LIN {X 0.129,Y -485.404,Z 1314.545,A 0.000,B 0.000,C 90.000,E1 98.106} C_DIS
LIN {X -0.160,Y -484.743,Z 1314.542,A 0.000,B 0.000,C 90.000,E1 97.644} C_DIS
LIN {X 0.035,Y -482.997,Z 1314.540,A 0.000,B 0.000,C 90.000,E1 97.125} C_DIS
LIN {X -0.080,Y -481.617,Z 1314.538,A 0.000,B 0.000,C 90.000,E1 96.891} C_DIS
LIN {X 0.196,Y -468.676,Z 1314.528,A 0.000,B 0.000,C 90.000,E1 95.106} C_DIS
LIN {X -0.021,Y -455.031,Z 1314.517,A 0.000,B 0.000,C 90.000,E1 93.094} C_DIS
LIN {X -0.140,Y -441.662,Z 1314.506,A 0.000,B 0.000,C 90.000,E1 91.031} C_DIS
LIN {X 0.133,Y -422.329,Z 1314.486,A 0.000,B 0.000,C 90.000,E1 87.535} C_DIS
LIN {X 0.147,Y -410.730,Z 1314.474,A 0.000,B 0.000,C 90.000,E1 85.355} C_DIS
LIN {X -0.079,Y -400.504,Z 1314.464,A 0.000,B 0.000,C 90.000,E1 83.451} C_DIS
LIN {X -0.116,Y -390.001,Z 1314.453,A 0.000,B 0.000,C 90.000,E1 81.489} C_DIS
LIN {X 0.060,Y -382.304,Z 1314.445,A 0.000,B 0.000,C 90.000,E1 80.038} C_DIS
LIN {X 0.190,Y -372.725,Z 1314.435,A 0.000,B 0.000,C 90.000,E1 78.285} C_DIS
LIN {X 0.196,Y -361.322,Z 1314.424,A 0.000,B 0.000,C 90.000,E1 76.228} C_DIS
LIN {X 0.053,Y -349.781,Z 1314.412,A 0.000,B 0.000,C 90.000,E1 74.157} C_DIS
LIN {X -0.138,Y -339.831,Z 1314.402,A 0.000,B 0.000,C 90.000,E1 72.362} C_DIS
LIN {X -0.137,Y -326.623,Z 1314.388,A 0.000,B 0.000,C 90.000,E1 69.880} C_DIS
LIN {X 0.035,Y -310.894,Z 1314.370,A 0.000,B 0.000,C 90.000,E1 66.666} C_DIS
LIN {X 0.081,Y -297.924,Z 1314.354,A 0.000,B 0.000,C 90.000,E1 63.717} C_DIS
LIN {X 0.082,Y -290.234,Z 1314.343,A 0.000,B 0.000,C 90.000,E1 61.719} C_DIS
LIN {X -0.050,Y -282.326,Z 1314.330,A 0.000,B 0.000,C 90.000,E1 59.380} C_DIS
LIN {X 0.051,Y -272.343,Z 1314.311,A 0.000,B 0.000,C 90.000,E1 55.928} C_DIS
LIN {X 0.059,Y -263.219,Z 1314.291,A 0.000,B 0.000,C 90.000,E1 52.431} C_DIS
LIN {X -0.081,Y -256.340,Z 1314.276,A 0.000,B 0.000,C 90.000,E1 49.622} C_DIS
LIN {X -0.074,Y -249.674,Z 1314.260,A 0.000,B 0.000,C 90.000,E1 46.743} C_DIS
LIN {X -0.083,Y -241.652,Z 1314.239,A 0.000,B 0.000,C 90.000,E1 43.095} C_DIS
LIN {X 0.031,Y -234.237,Z 1314.219,A 0.000,B 0.000,C 90.000,E1 39.358} C_DIS
LIN {X 0.013,Y -227.695,Z 1314.198,A 0.000,B 0.000,C 90.000,E1 35.598} C_DIS
LIN {X -0.050,Y -222.189,Z 1314.177,A 0.000,B 0.000,C 90.000,E1 31.799} C_DIS
LIN {X 0.121,Y -217.581,Z 1314.155,A 0.000,B 0.000,C 90.000,E1 27.897} C_DIS
LIN {X 0.034,Y -213.697,Z 1314.134,A 0.000,B 0.000,C 90.000,E1 24.027} C_DIS
LIN {X -0.036,Y -210.214,Z 1314.112,A 0.000,B 0.000,C 90.000,E1 20.120} C_DIS
LIN {X 0.080,Y -207.058,Z 1314.090,A 0.000,B 0.000,C 90.000,E1 16.134} C_DIS
LIN {X 0.003,Y -204.286,Z 1314.068,A 0.000,B 0.000,C 90.000,E1 12.175} C_DIS
LIN {X 0.056,Y -201.522,Z 1314.041,A 0.000,B 0.000,C 90.000,E1 7.352} C_DIS
LIN {X 0.006,Y -199.312,Z 1314.005,A 0.000,B 0.000,C 90.000,E1 0.917} C_DIS
LIN {X 0.017,Y -199.411,Z 1313.957,A 0.000,B 0.000,C 90.000,E1 352.243} C_DIS
LIN {X 0.019,Y -201.511,Z 1313.926,A 0.000,B 0.000,C 90.000,E1 346.589} C_DIS
LIN {X 0.030,Y -204.619,Z 1313.899,A 0.000,B 0.000,C 90.000,E1 341.764} C_DIS
LIN {X 0.046,Y -209.021,Z 1313.872,A 0.000,B 0.000,C 90.000,E1 336.975} C_DIS
LIN {X -0.054,Y -213.620,Z 1313.850,A 0.000,B 0.000,C 90.000,E1 333.050} C_DIS
LIN {X 0.001,Y -219.164,Z 1313.828,A 0.000,B 0.000,C 90.000,E1 329.125} C_DIS
LIN {X 0.001,Y -225.693,Z 1313.807,A 0.000,B 0.000,C 90.000,E1 325.261} C_DIS
LIN {X -0.020,Y -233.132,Z 1313.786,A 0.000,B 0.000,C 90.000,E1 321.457} C_DIS
LIN {X -0.056,Y -241.637,Z 1313.765,A 0.000,B 0.000,C 90.000,E1 317.715} C_DIS
LIN {X 0.140,Y -250.446,Z 1313.747,A 0.000,B 0.000,C 90.000,E1 314.352} C_DIS
LIN {X 0.079,Y -259.281,Z 1313.730,A 0.000,B 0.000,C 90.000,E1 311.472} C_DIS
LIN {X 0.033,Y -268.239,Z 1313.717,A 0.000,B 0.000,C 90.000,E1 308.991} C_DIS
LIN {X 0.134,Y -276.833,Z 1313.705,A 0.000,B 0.000,C 90.000,E1 306.870} C_DIS
LIN {X 0.035,Y -288.162,Z 1313.692,A 0.000,B 0.000,C 90.000,E1 304.485} C_DIS
LIN {X 0.018,Y -300.990,Z 1313.679,A 0.000,B 0.000,C 90.000,E1 302.133} C_DIS
LIN {X 0.100,Y -309.231,Z 1313.671,A 0.000,B 0.000,C 90.000,E1 300.797} C_DIS
LIN {X -0.073,Y -320.445,Z 1313.662,A 0.000,B 0.000,C 90.000,E1 299.205} C_DIS
LIN {X 0.014,Y -342.874,Z 1313.646,A 0.000,B 0.000,C 90.000,E1 296.360} C_DIS
LIN {X 0.027,Y -355.915,Z 1313.638,A 0.000,B 0.000,C 90.000,E1 294.847} C_DIS
LIN {X -0.173,Y -368.940,Z 1313.630,A 0.000,B 0.000,C 90.000,E1 293.387} C_DIS
LIN {X 0.041,Y -381.463,Z 1313.622,A 0.000,B 0.000,C 90.000,E1 291.897} C_DIS
LIN {X 0.046,Y -395.933,Z 1313.612,A 0.000,B 0.000,C 90.000,E1 290.174} C_DIS
LIN {X -0.031,Y -413.228,Z 1313.601,A 0.000,B 0.000,C 90.000,E1 288.236} C_DIS
LIN {X -0.116,Y -422.980,Z 1313.595,A 0.000,B 0.000,C 90.000,E1 287.149} C_DIS
LIN {X 0.037,Y -430.024,Z 1313.591,A 0.000,B 0.000,C 90.000,E1 286.315} C_DIS
LIN {X -0.180,Y -436.359,Z 1313.586,A 0.000,B 0.000,C 90.000,E1 285.552} C_DIS
LIN {X 0.104,Y -442.119,Z 1313.582,A 0.000,B 0.000,C 90.000,E1 284.717} C_DIS
LIN {X 0.003,Y -447.129,Z 1313.577,A 0.000,B 0.000,C 90.000,E1 283.939} C_DIS
LIN {X -0.161,Y -451.538,Z 1313.573,A 0.000,B 0.000,C 90.000,E1 283.175} C_DIS
LIN {X 0.153,Y -455.390,Z 1313.569,A 0.000,B 0.000,C 90.000,E1 282.355} C_DIS
LIN {X 0.237,Y -457.660,Z 1313.566,A 0.000,B 0.000,C 90.000,E1 281.827} C_DIS
LIN {X -0.206,Y -459.677,Z 1313.563,A 0.000,B 0.000,C 90.000,E1 281.366} C_DIS
LIN {X -0.102,Y -461.296,Z 1313.560,A 0.000,B 0.000,C 90.000,E1 280.838} C_DIS
LIN {X 0.014,Y -462.553,Z 1313.557,A 0.000,B 0.000,C 90.000,E1 280.310} C_DIS
LIN {X 0.057,Y -463.410,Z 1313.554,A 0.000,B 0.000,C 90.000,E1 279.792} C_DIS
LIN {X 0.186,Y -463.807,Z 1313.552,A 0.000,B 0.000,C 90.000,E1 279.265} C_DIS
LIN {X -0.213,Y -463.825,Z 1313.549,A 0.000,B 0.000,C 90.000,E1 278.803} C_DIS
LIN {X -0.082,Y -463.391,Z 1313.546,A 0.000,B 0.000,C 90.000,E1 278.276} C_DIS
LIN {X -0.018,Y -462.473,Z 1313.543,A 0.000,B 0.000,C 90.000,E1 277.757} C_DIS
LIN {X 0.043,Y -461.050,Z 1313.540,A 0.000,B 0.000,C 90.000,E1 277.239} C_DIS
LIN {X 0.100,Y -459.176,Z 1313.537,A 0.000,B 0.000,C 90.000,E1 276.720} C_DIS
LIN {X 0.150,Y -456.758,Z 1313.535,A 0.000,B 0.000,C 90.000,E1 276.201} C_DIS
LIN {X 0.180,Y -453.846,Z 1313.532,A 0.000,B 0.000,C 90.000,E1 275.682} C_DIS
LIN {X 0.194,Y -450.298,Z 1313.529,A 0.000,B 0.000,C 90.000,E1 275.163} C_DIS
LIN {X 0.189,Y -446.103,Z 1313.526,A 0.000,B 0.000,C 90.000,E1 274.645} C_DIS
LIN {X 0.126,Y -440.950,Z 1313.523,A 0.000,B 0.000,C 90.000,E1 274.131} C_DIS
LIN {X -0.144,Y -435.047,Z 1313.520,A 0.000,B 0.000,C 90.000,E1 273.669} C_DIS
LIN {X -0.034,Y -428.759,Z 1313.518,A 0.000,B 0.000,C 90.000,E1 273.212} C_DIS
LIN {X 0.099,Y -422.212,Z 1313.516,A 0.000,B 0.000,C 90.000,E1 272.808} C_DIS
LIN {X 0.175,Y -415.466,Z 1313.514,A 0.000,B 0.000,C 90.000,E1 272.465} C_DIS
LIN {X 0.182,Y -408.449,Z 1313.512,A 0.000,B 0.000,C 90.000,E1 272.178} C_DIS
LIN {X 0.125,Y -401.313,Z 1313.511,A 0.000,B 0.000,C 90.000,E1 271.949} C_DIS
LIN {X 0.192,Y -390.679,Z 1313.509,A 0.000,B 0.000,C 90.000,E1 271.661} C_DIS
LIN {X -0.029,Y -382.994,Z 1313.509,A 0.000,B 0.000,C 90.000,E1 271.547} C_DIS
LIN {X -0.046,Y -374.676,Z 1313.508,A 0.000,B 0.000,C 90.000,E1 271.432} C_DIS
LIN {X 0.106,Y -362.236,Z 1313.507,A 0.000,B 0.000,C 90.000,E1 271.318} C_DIS
LIN {X -0.135,Y -348.212,Z 1313.507,A 0.000,B 0.000,C 90.000,E1 271.318} C_DIS
LIN {X 0.075,Y -181.395,Z 1313.507,A 0.000,B 0.000,C 90.000,E1 271.260} C_DIS
LIN {X 0.024,Y -181.576,Z 1313.502,A 0.000,B 0.000,C 90.000,E1 270.401} C_DIS
LIN {X 0.000,Y -180.906,Z 1313.474,A 0.000,B 0.000,C 90.000,E1 265.355} C_DIS
LIN {X 0.074,Y -180.682,Z 1313.469,A 0.000,B 0.000,C 90.000,E1 264.489} C_DIS
LIN {X -0.028,Y -178.765,Z 1313.441,A 0.000,B 0.000,C 90.000,E1 259.454} C_DIS
LIN {X 0.044,Y -175.812,Z 1313.413,A 0.000,B 0.000,C 90.000,E1 254.338} C_DIS
LIN {X 0.038,Y -171.997,Z 1313.385,A 0.000,B 0.000,C 90.000,E1 249.209} C_DIS
LIN {X 0.013,Y -171.411,Z 1313.380,A 0.000,B 0.000,C 90.000,E1 248.358} C_DIS
LIN {X 0.060,Y -167.651,Z 1313.356,A 0.000,B 0.000,C 90.000,E1 244.024} C_DIS
LIN {X 0.076,Y -166.316,Z 1313.346,A 0.000,B 0.000,C 90.000,E1 242.281} C_DIS
LIN {X 0.068,Y -163.058,Z 1313.327,A 0.000,B 0.000,C 90.000,E1 238.791} C_DIS
LIN {X 0.030,Y -160.993,Z 1313.312,A 0.000,B 0.000,C 90.000,E1 236.167} C_DIS
LIN {X 0.007,Y -157.740,Z 1313.292,A 0.000,B 0.000,C 90.000,E1 232.637} C_DIS
LIN {X -0.055,Y -155.779,Z 1313.278,A 0.000,B 0.000,C 90.000,E1 229.989} C_DIS
LIN {X 0.001,Y -152.033,Z 1313.253,A 0.000,B 0.000,C 90.000,E1 225.486} C_DIS
LIN {X 0.018,Y -150.282,Z 1313.238,A 0.000,B 0.000,C 90.000,E1 222.771} C_DIS
LIN {X -0.055,Y -147.031,Z 1313.212,A 0.000,B 0.000,C 90.000,E1 218.257} C_DIS
LIN {X -0.062,Y -145.612,Z 1313.197,A 0.000,B 0.000,C 90.000,E1 215.518} C_DIS
LIN {X -0.063,Y -142.997,Z 1313.172,A 0.000,B 0.000,C 90.000,E1 210.924} C_DIS
LIN {X -0.006,Y -141.624,Z 1313.151,A 0.000,B 0.000,C 90.000,E1 207.206} C_DIS
LIN {X -0.080,Y -139.433,Z 1313.115,A 0.000,B 0.000,C 90.000,E1 200.737} C_DIS
LIN {X -0.026,Y -139.164,Z 1313.105,A 0.000,B 0.000,C 90.000,E1 198.852} C_DIS
LIN {X 0.012,Y -138.340,Z 1313.058,A 0.000,B 0.000,C 90.000,E1 190.433} C_DIS
LIN {X 0.019,Y -139.478,Z 1313.006,A 0.000,B 0.000,C 90.000,E1 181.088} C_DIS
LIN {X -0.041,Y -141.062,Z 1312.975,A 0.000,B 0.000,C 90.000,E1 175.527} C_DIS
LIN {X 0.054,Y -142.435,Z 1312.960,A 0.000,B 0.000,C 90.000,E1 172.704} C_DIS
LIN {X -0.026,Y -144.674,Z 1312.934,A 0.000,B 0.000,C 90.000,E1 168.117} C_DIS
LIN {X -0.043,Y -147.261,Z 1312.913,A 0.000,B 0.000,C 90.000,E1 164.448} C_DIS
LIN {X -0.026,Y -150.578,Z 1312.888,A 0.000,B 0.000,C 90.000,E1 159.880} C_DIS
LIN {X 0.053,Y -154.049,Z 1312.868,A 0.000,B 0.000,C 90.000,E1 156.230} C_DIS
LIN {X -0.020,Y -157.466,Z 1312.848,A 0.000,B 0.000,C 90.000,E1 152.666} C_DIS
LIN {X 0.067,Y -161.688,Z 1312.828,A 0.000,B 0.000,C 90.000,E1 149.076} C_DIS
LIN {X -0.055,Y -165.882,Z 1312.809,A 0.000,B 0.000,C 90.000,E1 145.595} C_DIS
LIN {X -0.065,Y -170.864,Z 1312.789,A 0.000,B 0.000,C 90.000,E1 142.110} C_DIS
LIN {X -0.018,Y -175.732,Z 1312.770,A 0.000,B 0.000,C 90.000,E1 138.647} C_DIS
LIN {X -0.028,Y -181.343,Z 1312.751,A 0.000,B 0.000,C 90.000,E1 135.243} C_DIS
LIN {X 0.106,Y -186.832,Z 1312.733,A 0.000,B 0.000,C 90.000,E1 131.838} C_DIS
LIN {X 0.060,Y -191.419,Z 1312.719,A 0.000,B 0.000,C 90.000,E1 129.358} C_DIS
LIN {X -0.007,Y -197.268,Z 1312.700,A 0.000,B 0.000,C 90.000,E1 126.091} C_DIS
LIN {X 0.100,Y -199.328,Z 1312.695,A 0.000,B 0.000,C 90.000,E1 125.025} C_DIS
LIN {X 0.108,Y -309.118,Z 1312.695,A 0.000,B 0.000,C 90.000,E1 125.025} C_DIS
LIN {X -0.037,Y -310.705,Z 1312.695,A 0.000,B 0.000,C 90.000,E1 125.025} C_DIS
LIN {X 0.004,Y -316.189,Z 1312.693,A 0.000,B 0.000,C 90.000,E1 124.739} C_DIS
LIN {X 0.047,Y -319.053,Z 1312.691,A 0.000,B 0.000,C 90.000,E1 124.452} C_DIS
LIN {X 0.004,Y -322.705,Z 1312.688,A 0.000,B 0.000,C 90.000,E1 123.913} C_DIS
LIN {X 0.083,Y -324.185,Z 1312.687,A 0.000,B 0.000,C 90.000,E1 123.579} C_DIS
LIN {X -0.004,Y -337.025,Z 1312.667,A 0.000,B 0.000,C 90.000,E1 120.129} C_DIS
LIN {X 0.111,Y -348.953,Z 1312.652,A 0.000,B 0.000,C 90.000,E1 117.334} C_DIS
LIN {X -0.069,Y -362.342,Z 1312.637,A 0.000,B 0.000,C 90.000,E1 114.643} C_DIS
LIN {X -0.098,Y -375.559,Z 1312.624,A 0.000,B 0.000,C 90.000,E1 112.280} C_DIS
LIN {X 0.068,Y -390.111,Z 1312.611,A 0.000,B 0.000,C 90.000,E1 109.939} C_DIS
LIN {X -0.044,Y -406.099,Z 1312.598,A 0.000,B 0.000,C 90.000,E1 107.692} C_DIS
LIN {X -0.017,Y -423.638,Z 1312.586,A 0.000,B 0.000,C 90.000,E1 105.481} C_DIS
LIN {X -0.171,Y -442.816,Z 1312.574,A 0.000,B 0.000,C 90.000,E1 103.355} C_DIS
LIN {X 0.255,Y -462.921,Z 1312.563,A 0.000,B 0.000,C 90.000,E1 101.299} C_DIS
LIN {X -0.217,Y -478.305,Z 1312.555,A 0.000,B 0.000,C 90.000,E1 99.962} C_DIS
LIN {X -0.161,Y -480.341,Z 1312.554,A 0.000,B 0.000,C 90.000,E1 99.726} C_DIS
LIN {X -0.186,Y -481.890,Z 1312.553,A 0.000,B 0.000,C 90.000,E1 99.500} C_DIS
LIN {X 0.171,Y -483.176,Z 1312.551,A 0.000,B 0.000,C 90.000,E1 99.208} C_DIS
LIN {X 0.051,Y -484.119,Z 1312.550,A 0.000,B 0.000,C 90.000,E1 98.973} C_DIS
LIN {X 0.229,Y -485.156,Z 1312.547,A 0.000,B 0.000,C 90.000,E1 98.454} C_DIS
LIN {X -0.065,Y -485.192,Z 1312.544,A 0.000,B 0.000,C 90.000,E1 97.992} C_DIS
LIN {X 0.129,Y -484.236,Z 1312.542,A 0.000,B 0.000,C 90.000,E1 97.473} C_DIS
LIN {X -0.096,Y -482.124,Z 1312.539,A 0.000,B 0.000,C 90.000,E1 97.004} C_DIS
LIN {X 0.206,Y -480.494,Z 1312.537,A 0.000,B 0.000,C 90.000,E1 96.720} C_DIS
LIN {X 0.187,Y -469.256,Z 1312.529,A 0.000,B 0.000,C 90.000,E1 95.220} C_DIS
LIN {X -0.045,Y -455.588,Z 1312.518,A 0.000,B 0.000,C 90.000,E1 93.212} C_DIS
LIN {X -0.126,Y -442.157,Z 1312.506,A 0.000,B 0.000,C 90.000,E1 91.146} C_DIS
LIN {X 0.168,Y -422.747,Z 1312.487,A 0.000,B 0.000,C 90.000,E1 87.650} C_DIS
LIN {X 0.108,Y -412.604,Z 1312.476,A 0.000,B 0.000,C 90.000,E1 85.755} C_DIS
LIN {X 0.189,Y -403.883,Z 1312.467,A 0.000,B 0.000,C 90.000,E1 84.090} C_DIS
LIN {X 0.196,Y -394.970,Z 1312.458,A 0.000,B 0.000,C 90.000,E1 82.413} C_DIS
LIN {X 0.049,Y -385.900,Z 1312.449,A 0.000,B 0.000,C 90.000,E1 80.735} C_DIS
LIN {X 0.156,Y -378.059,Z 1312.441,A 0.000,B 0.000,C 90.000,E1 79.285} C_DIS
LIN {X -0.158,Y -368.373,Z 1312.431,A 0.000,B 0.000,C 90.000,E1 77.589} C_DIS
LIN {X -0.112,Y -358.566,Z 1312.421,A 0.000,B 0.000,C 90.000,E1 75.811} C_DIS
LIN {X 0.102,Y -348.668,Z 1312.411,A 0.000,B 0.000,C 90.000,E1 73.976} C_DIS
LIN {X -0.109,Y -338.711,Z 1312.401,A 0.000,B 0.000,C 90.000,E1 72.181} C_DIS
LIN {X -0.137,Y -325.538,Z 1312.387,A 0.000,B 0.000,C 90.000,E1 69.699} C_DIS
LIN {X 0.000,Y -309.901,Z 1312.369,A 0.000,B 0.000,C 90.000,E1 66.485} C_DIS
LIN {X 0.147,Y -297.056,Z 1312.353,A 0.000,B 0.000,C 90.000,E1 63.512} C_DIS
LIN {X 0.136,Y -289.470,Z 1312.342,A 0.000,B 0.000,C 90.000,E1 61.513} C_DIS
LIN {X -0.155,Y -281.660,Z 1312.329,A 0.000,B 0.000,C 90.000,E1 59.203} C_DIS
LIN {X 0.071,Y -271.755,Z 1312.310,A 0.000,B 0.000,C 90.000,E1 55.722} C_DIS
LIN {X -0.150,Y -262.678,Z 1312.290,A 0.000,B 0.000,C 90.000,E1 52.271} C_DIS
LIN {X 0.067,Y -255.828,Z 1312.274,A 0.000,B 0.000,C 90.000,E1 49.380} C_DIS
LIN {X -0.110,Y -249.157,Z 1312.258,A 0.000,B 0.000,C 90.000,E1 46.539} C_DIS
LIN {X 0.031,Y -241.153,Z 1312.238,A 0.000,B 0.000,C 90.000,E1 42.852} C_DIS
LIN {X 0.121,Y -233.760,Z 1312.218,A 0.000,B 0.000,C 90.000,E1 39.116} C_DIS
LIN {X -0.054,Y -227.286,Z 1312.197,A 0.000,B 0.000,C 90.000,E1 35.391} C_DIS
LIN {X 0.063,Y -221.831,Z 1312.175,A 0.000,B 0.000,C 90.000,E1 31.544} C_DIS
LIN {X -0.071,Y -217.244,Z 1312.154,A 0.000,B 0.000,C 90.000,E1 27.719} C_DIS
LIN {X -0.072,Y -213.324,Z 1312.132,A 0.000,B 0.000,C 90.000,E1 23.823} C_DIS
LIN {X -0.037,Y -209.863,Z 1312.110,A 0.000,B 0.000,C 90.000,E1 19.885} C_DIS
LIN {X 0.071,Y -206.677,Z 1312.088,A 0.000,B 0.000,C 90.000,E1 15.898} C_DIS
LIN {X -0.059,Y -203.896,Z 1312.066,A 0.000,B 0.000,C 90.000,E1 11.951} C_DIS
LIN {X 0.011,Y -200.828,Z 1312.035,A 0.000,B 0.000,C 90.000,E1 6.315} C_DIS
LIN {X -0.036,Y -198.918,Z 1311.997,A 0.000,B 0.000,C 90.000,E1 359.542} C_DIS
LIN {X 0.056,Y -200.020,Z 1311.943,A 0.000,B 0.000,C 90.000,E1 349.803} C_DIS
LIN {X 0.065,Y -202.851,Z 1311.912,A 0.000,B 0.000,C 90.000,E1 344.157} C_DIS
LIN {X -0.073,Y -206.696,Z 1311.885,A 0.000,B 0.000,C 90.000,E1 339.390} C_DIS
LIN {X -0.041,Y -210.815,Z 1311.863,A 0.000,B 0.000,C 90.000,E1 335.409} C_DIS
LIN {X -0.001,Y -215.800,Z 1311.841,A 0.000,B 0.000,C 90.000,E1 331.463} C_DIS
LIN {X -0.043,Y -221.742,Z 1311.820,A 0.000,B 0.000,C 90.000,E1 327.582} C_DIS
LIN {X 0.101,Y -228.659,Z 1311.798,A 0.000,B 0.000,C 90.000,E1 323.703} C_DIS
LIN {X 0.141,Y -236.482,Z 1311.777,A 0.000,B 0.000,C 90.000,E1 319.908} C_DIS
LIN {X 0.058,Y -243.554,Z 1311.761,A 0.000,B 0.000,C 90.000,E1 316.944} C_DIS
LIN {X 0.141,Y -252.614,Z 1311.743,A 0.000,B 0.000,C 90.000,E1 313.623} C_DIS
LIN {X -0.084,Y -260.533,Z 1311.729,A 0.000,B 0.000,C 90.000,E1 311.148} C_DIS
LIN {X -0.109,Y -269.636,Z 1311.715,A 0.000,B 0.000,C 90.000,E1 308.669} C_DIS
LIN {X -0.157,Y -278.420,Z 1311.703,A 0.000,B 0.000,C 90.000,E1 306.583} C_DIS
LIN {X 0.034,Y -288.204,Z 1311.692,A 0.000,B 0.000,C 90.000,E1 304.485} C_DIS
LIN {X 0.018,Y -301.049,Z 1311.679,A 0.000,B 0.000,C 90.000,E1 302.133} C_DIS
LIN {X 0.101,Y -309.297,Z 1311.671,A 0.000,B 0.000,C 90.000,E1 300.797} C_DIS
LIN {X -0.139,Y -318.164,Z 1311.664,A 0.000,B 0.000,C 90.000,E1 299.539} C_DIS
LIN {X 0.169,Y -335.277,Z 1311.652,A 0.000,B 0.000,C 90.000,E1 297.257} C_DIS
LIN {X -0.172,Y -353.539,Z 1311.640,A 0.000,B 0.000,C 90.000,E1 295.155} C_DIS
LIN {X -0.100,Y -366.593,Z 1311.631,A 0.000,B 0.000,C 90.000,E1 293.643} C_DIS
LIN {X 0.039,Y -379.295,Z 1311.623,A 0.000,B 0.000,C 90.000,E1 292.153} C_DIS
LIN {X -0.072,Y -391.293,Z 1311.615,A 0.000,B 0.000,C 90.000,E1 290.737} C_DIS
LIN {X -0.101,Y -411.032,Z 1311.603,A 0.000,B 0.000,C 90.000,E1 288.489} C_DIS
LIN {X 0.066,Y -423.259,Z 1311.595,A 0.000,B 0.000,C 90.000,E1 287.094} C_DIS
LIN {X -0.187,Y -430.279,Z 1311.590,A 0.000,B 0.000,C 90.000,E1 286.315} C_DIS
LIN {X 0.027,Y -436.718,Z 1311.586,A 0.000,B 0.000,C 90.000,E1 285.481} C_DIS
LIN {X -0.228,Y -442.417,Z 1311.582,A 0.000,B 0.000,C 90.000,E1 284.717} C_DIS
LIN {X 0.105,Y -447.375,Z 1311.577,A 0.000,B 0.000,C 90.000,E1 283.883} C_DIS
LIN {X -0.055,Y -451.670,Z 1311.573,A 0.000,B 0.000,C 90.000,E1 283.119} C_DIS
LIN {X -0.183,Y -455.501,Z 1311.568,A 0.000,B 0.000,C 90.000,E1 282.355} C_DIS
LIN {X -0.099,Y -457.778,Z 1311.566,A 0.000,B 0.000,C 90.000,E1 281.827} C_DIS
LIN {X -0.002,Y -459.785,Z 1311.563,A 0.000,B 0.000,C 90.000,E1 281.299} C_DIS
LIN {X 0.015,Y -461.400,Z 1311.560,A 0.000,B 0.000,C 90.000,E1 280.782} C_DIS
LIN {X 0.131,Y -462.631,Z 1311.557,A 0.000,B 0.000,C 90.000,E1 280.254} C_DIS
LIN {X 0.254,Y -463.511,Z 1311.554,A 0.000,B 0.000,C 90.000,E1 279.726} C_DIS
LIN {X -0.152,Y -463.900,Z 1311.551,A 0.000,B 0.000,C 90.000,E1 279.265} C_DIS
LIN {X -0.091,Y -463.943,Z 1311.549,A 0.000,B 0.000,C 90.000,E1 278.746} C_DIS
LIN {X 0.041,Y -463.510,Z 1311.546,A 0.000,B 0.000,C 90.000,E1 278.219} C_DIS
LIN {X 0.105,Y -462.590,Z 1311.543,A 0.000,B 0.000,C 90.000,E1 277.701} C_DIS
LIN {X 0.168,Y -461.190,Z 1311.540,A 0.000,B 0.000,C 90.000,E1 277.182} C_DIS
LIN {X -0.230,Y -459.312,Z 1311.537,A 0.000,B 0.000,C 90.000,E1 276.720} C_DIS
LIN {X -0.179,Y -456.893,Z 1311.534,A 0.000,B 0.000,C 90.000,E1 276.201} C_DIS
LIN {X -0.145,Y -453.966,Z 1311.531,A 0.000,B 0.000,C 90.000,E1 275.682} C_DIS
LIN {X -0.128,Y -450.443,Z 1311.529,A 0.000,B 0.000,C 90.000,E1 275.163} C_DIS
LIN {X -0.130,Y -446.269,Z 1311.526,A 0.000,B 0.000,C 90.000,E1 274.645} C_DIS
LIN {X -0.188,Y -441.118,Z 1311.523,A 0.000,B 0.000,C 90.000,E1 274.131} C_DIS
LIN {X 0.002,Y -435.278,Z 1311.520,A 0.000,B 0.000,C 90.000,E1 273.612} C_DIS
LIN {X 0.121,Y -428.979,Z 1311.518,A 0.000,B 0.000,C 90.000,E1 273.154} C_DIS
LIN {X -0.181,Y -422.422,Z 1311.516,A 0.000,B 0.000,C 90.000,E1 272.808} C_DIS
LIN {X -0.101,Y -415.686,Z 1311.514,A 0.000,B 0.000,C 90.000,E1 272.465} C_DIS
LIN {X -0.109,Y -408.550,Z 1311.512,A 0.000,B 0.000,C 90.000,E1 272.178} C_DIS
LIN {X -0.154,Y -401.365,Z 1311.511,A 0.000,B 0.000,C 90.000,E1 271.949} C_DIS
LIN {X -0.075,Y -390.415,Z 1311.509,A 0.000,B 0.000,C 90.000,E1 271.661} C_DIS
LIN {X 0.095,Y -382.732,Z 1311.508,A 0.000,B 0.000,C 90.000,E1 271.489} C_DIS
LIN {X 0.092,Y -373.920,Z 1311.508,A 0.000,B 0.000,C 90.000,E1 271.375} C_DIS
LIN {X 0.015,Y -365.346,Z 1311.507,A 0.000,B 0.000,C 90.000,E1 271.318} C_DIS
LIN {X 0.069,Y -350.108,Z 1311.507,A 0.000,B 0.000,C 90.000,E1 271.260} C_DIS
LIN {X 0.005,Y -181.399,Z 1311.507,A 0.000,B 0.000,C 90.000,E1 271.260} C_DIS
LIN {X 0.049,Y -181.581,Z 1311.501,A 0.000,B 0.000,C 90.000,E1 270.229} C_DIS
LIN {X 0.053,Y -180.867,Z 1311.472,A 0.000,B 0.000,C 90.000,E1 265.008} C_DIS
LIN {X -0.070,Y -178.982,Z 1311.444,A 0.000,B 0.000,C 90.000,E1 259.982} C_DIS
LIN {X -0.058,Y -177.954,Z 1311.435,A 0.000,B 0.000,C 90.000,E1 258.285} C_DIS
LIN {X -0.039,Y -175.596,Z 1311.411,A 0.000,B 0.000,C 90.000,E1 254.031} C_DIS
LIN {X -0.027,Y -172.321,Z 1311.387,A 0.000,B 0.000,C 90.000,E1 249.752} C_DIS
LIN {X -0.047,Y -171.799,Z 1311.383,A 0.000,B 0.000,C 90.000,E1 248.901} C_DIS
LIN {X -0.010,Y -169.471,Z 1311.368,A 0.000,B 0.000,C 90.000,E1 246.305} C_DIS
LIN {X 0.046,Y -166.798,Z 1311.349,A 0.000,B 0.000,C 90.000,E1 242.820} C_DIS
LIN {X 0.040,Y -162.779,Z 1311.325,A 0.000,B 0.000,C 90.000,E1 238.456} C_DIS
LIN {X 0.016,Y -161.468,Z 1311.315,A 0.000,B 0.000,C 90.000,E1 236.707} C_DIS
LIN {X 0.057,Y -157.463,Z 1311.291,A 0.000,B 0.000,C 90.000,E1 232.271} C_DIS
LIN {X -0.010,Y -155.475,Z 1311.276,A 0.000,B 0.000,C 90.000,E1 229.622} C_DIS
LIN {X -0.077,Y -151.786,Z 1311.251,A 0.000,B 0.000,C 90.000,E1 225.162} C_DIS
LIN {X -0.063,Y -149.993,Z 1311.236,A 0.000,B 0.000,C 90.000,E1 222.447} C_DIS
LIN {X -0.033,Y -146.824,Z 1311.210,A 0.000,B 0.000,C 90.000,E1 217.890} C_DIS
LIN {X 0.074,Y -145.403,Z 1311.195,A 0.000,B 0.000,C 90.000,E1 215.105} C_DIS
LIN {X -0.009,Y -142.836,Z 1311.170,A 0.000,B 0.000,C 90.000,E1 210.541} C_DIS
LIN {X -0.079,Y -141.449,Z 1311.149,A 0.000,B 0.000,C 90.000,E1 206.873} C_DIS
LIN {X -0.039,Y -139.371,Z 1311.113,A 0.000,B 0.000,C 90.000,E1 200.355} C_DIS
LIN {X 0.036,Y -138.820,Z 1311.097,A 0.000,B 0.000,C 90.000,E1 197.528} C_DIS
LIN {X -0.009,Y -138.353,Z 1311.056,A 0.000,B 0.000,C 90.000,E1 190.074} C_DIS
LIN {X -0.035,Y -139.534,Z 1311.004,A 0.000,B 0.000,C 90.000,E1 180.745} C_DIS
LIN {X 0.058,Y -141.220,Z 1310.973,A 0.000,B 0.000,C 90.000,E1 175.122} C_DIS
LIN {X 0.017,Y -142.593,Z 1310.958,A 0.000,B 0.000,C 90.000,E1 172.356} C_DIS
LIN {X -0.030,Y -144.895,Z 1310.932,A 0.000,B 0.000,C 90.000,E1 167.757} C_DIS
LIN {X -0.076,Y -147.523,Z 1310.911,A 0.000,B 0.000,C 90.000,E1 164.102} C_DIS
LIN {X -0.002,Y -150.119,Z 1310.891,A 0.000,B 0.000,C 90.000,E1 160.423} C_DIS
LIN {X 0.010,Y -153.480,Z 1310.871,A 0.000,B 0.000,C 90.000,E1 156.794} C_DIS
LIN {X 0.073,Y -157.844,Z 1310.846,A 0.000,B 0.000,C 90.000,E1 152.281} C_DIS
LIN {X 0.029,Y -162.128,Z 1310.826,A 0.000,B 0.000,C 90.000,E1 148.742} C_DIS
LIN {X 0.009,Y -166.332,Z 1310.807,A 0.000,B 0.000,C 90.000,E1 145.229} C_DIS
LIN {X 0.016,Y -171.349,Z 1310.787,A 0.000,B 0.000,C 90.000,E1 141.743} C_DIS
LIN {X -0.057,Y -176.252,Z 1310.768,A 0.000,B 0.000,C 90.000,E1 138.324} C_DIS
LIN {X 0.062,Y -180.535,Z 1310.754,A 0.000,B 0.000,C 90.000,E1 135.729} C_DIS
LIN {X 0.041,Y -185.937,Z 1310.735,A 0.000,B 0.000,C 90.000,E1 132.366} C_DIS
LIN {X -0.024,Y -190.567,Z 1310.722,A 0.000,B 0.000,C 90.000,E1 129.886} C_DIS
LIN {X 0.007,Y -196.317,Z 1310.703,A 0.000,B 0.000,C 90.000,E1 126.583} C_DIS
LIN {X 0.059,Y -199.352,Z 1310.695,A 0.000,B 0.000,C 90.000,E1 125.025} C_DIS
LIN {X 0.058,Y -308.896,Z 1310.695,A 0.000,B 0.000,C 90.000,E1 125.025} C_DIS
LIN {X 0.050,Y -312.366,Z 1310.694,A 0.000,B 0.000,C 90.000,E1 124.945} C_DIS
LIN {X 0.014,Y -315.602,Z 1310.693,A 0.000,B 0.000,C 90.000,E1 124.771} C_DIS
LIN {X 0.155,Y -319.210,Z 1310.691,A 0.000,B 0.000,C 90.000,E1 124.405} C_DIS
LIN {X -0.085,Y -322.744,Z 1310.688,A 0.000,B 0.000,C 90.000,E1 123.913} C_DIS
LIN {X -0.006,Y -324.221,Z 1310.687,A 0.000,B 0.000,C 90.000,E1 123.579} C_DIS
LIN {X -0.094,Y -337.066,Z 1310.667,A 0.000,B 0.000,C 90.000,E1 120.129} C_DIS
LIN {X 0.017,Y -349.001,Z 1310.652,A 0.000,B 0.000,C 90.000,E1 117.334} C_DIS
LIN {X -0.164,Y -362.398,Z 1310.637,A 0.000,B 0.000,C 90.000,E1 114.643} C_DIS
LIN {X -0.054,Y -375.623,Z 1310.624,A 0.000,B 0.000,C 90.000,E1 112.259} C_DIS
LIN {X -0.030,Y -390.183,Z 1310.611,A 0.000,B 0.000,C 90.000,E1 109.939} C_DIS
LIN {X -0.145,Y -406.180,Z 1310.598,A 0.000,B 0.000,C 90.000,E1 107.692} C_DIS
LIN {X -0.120,Y -423.729,Z 1310.586,A 0.000,B 0.000,C 90.000,E1 105.481} C_DIS
LIN {X 0.156,Y -442.917,Z 1310.574,A 0.000,B 0.000,C 90.000,E1 103.300} C_DIS
LIN {X 0.153,Y -463.025,Z 1310.563,A 0.000,B 0.000,C 90.000,E1 101.299} C_DIS
LIN {X 0.156,Y -478.383,Z 1310.555,A 0.000,B 0.000,C 90.000,E1 99.905} C_DIS
LIN {X 0.199,Y -480.378,Z 1310.554,A 0.000,B 0.000,C 90.000,E1 99.670} C_DIS
LIN {X 0.164,Y -481.900,Z 1310.553,A 0.000,B 0.000,C 90.000,E1 99.443} C_DIS
LIN {X 0.045,Y -483.150,Z 1310.551,A 0.000,B 0.000,C 90.000,E1 99.208} C_DIS
LIN {X -0.075,Y -484.065,Z 1310.550,A 0.000,B 0.000,C 90.000,E1 98.973} C_DIS
LIN {X 0.103,Y -485.054,Z 1310.547,A 0.000,B 0.000,C 90.000,E1 98.454} C_DIS
LIN {X -0.191,Y -485.047,Z 1310.544,A 0.000,B 0.000,C 90.000,E1 97.992} C_DIS
LIN {X 0.065,Y -484.044,Z 1310.542,A 0.000,B 0.000,C 90.000,E1 97.466} C_DIS
LIN {X -0.110,Y -483.125,Z 1310.540,A 0.000,B 0.000,C 90.000,E1 97.239} C_DIS
LIN {X 0.255,Y -481.871,Z 1310.539,A 0.000,B 0.000,C 90.000,E1 96.947} C_DIS
LIN {X 0.076,Y -480.196,Z 1310.537,A 0.000,B 0.000,C 90.000,E1 96.720} C_DIS
LIN {X 0.052,Y -468.950,Z 1310.529,A 0.000,B 0.000,C 90.000,E1 95.220} C_DIS
LIN {X -0.181,Y -455.270,Z 1310.518,A 0.000,B 0.000,C 90.000,E1 93.212} C_DIS
LIN {X -0.079,Y -440.258,Z 1310.505,A 0.000,B 0.000,C 90.000,E1 90.859} C_DIS
LIN {X 0.021,Y -422.422,Z 1310.487,A 0.000,B 0.000,C 90.000,E1 87.650} C_DIS
LIN {X 0.044,Y -410.866,Z 1310.475,A 0.000,B 0.000,C 90.000,E1 85.469} C_DIS
LIN {X 0.132,Y -402.108,Z 1310.466,A 0.000,B 0.000,C 90.000,E1 83.799} C_DIS
LIN {X 0.121,Y -391.678,Z 1310.455,A 0.000,B 0.000,C 90.000,E1 81.837} C_DIS
LIN {X -0.024,Y -382.501,Z 1310.445,A 0.000,B 0.000,C 90.000,E1 80.151} C_DIS
LIN {X 0.042,Y -372.944,Z 1310.436,A 0.000,B 0.000,C 90.000,E1 78.409} C_DIS
LIN {X 0.077,Y -363.211,Z 1310.426,A 0.000,B 0.000,C 90.000,E1 76.645} C_DIS
LIN {X -0.026,Y -351.683,Z 1310.414,A 0.000,B 0.000,C 90.000,E1 74.574} C_DIS
LIN {X 0.151,Y -340.068,Z 1310.402,A 0.000,B 0.000,C 90.000,E1 72.417} C_DIS
LIN {X 0.150,Y -326.864,Z 1310.389,A 0.000,B 0.000,C 90.000,E1 69.934} C_DIS
LIN {X -0.087,Y -311.185,Z 1310.371,A 0.000,B 0.000,C 90.000,E1 66.794} C_DIS
LIN {X -0.024,Y -298.194,Z 1310.355,A 0.000,B 0.000,C 90.000,E1 63.845} C_DIS
LIN {X -0.015,Y -290.488,Z 1310.344,A 0.000,B 0.000,C 90.000,E1 61.847} C_DIS
LIN {X 0.070,Y -281.511,Z 1310.328,A 0.000,B 0.000,C 90.000,E1 59.125} C_DIS
LIN {X -0.088,Y -271.626,Z 1310.309,A 0.000,B 0.000,C 90.000,E1 55.722} C_DIS
LIN {X 0.061,Y -262.564,Z 1310.290,A 0.000,B 0.000,C 90.000,E1 52.190} C_DIS
LIN {X -0.089,Y -255.714,Z 1310.274,A 0.000,B 0.000,C 90.000,E1 49.380} C_DIS
LIN {X 0.086,Y -249.019,Z 1310.258,A 0.000,B 0.000,C 90.000,E1 46.458} C_DIS
LIN {X 0.071,Y -242.567,Z 1310.242,A 0.000,B 0.000,C 90.000,E1 43.542} C_DIS
LIN {X 0.025,Y -235.024,Z 1310.221,A 0.000,B 0.000,C 90.000,E1 39.850} C_DIS
LIN {X 0.024,Y -228.382,Z 1310.201,A 0.000,B 0.000,C 90.000,E1 36.091} C_DIS
LIN {X -0.015,Y -222.709,Z 1310.179,A 0.000,B 0.000,C 90.000,E1 32.291} C_DIS
LIN {X -0.009,Y -217.943,Z 1310.158,A 0.000,B 0.000,C 90.000,E1 28.437} C_DIS
LIN {X 0.105,Y -213.890,Z 1310.136,A 0.000,B 0.000,C 90.000,E1 24.515} C_DIS
LIN {X 0.071,Y -209.634,Z 1310.110,A 0.000,B 0.000,C 90.000,E1 19.812} C_DIS
LIN {X 0.103,Y -206.416,Z 1310.088,A 0.000,B 0.000,C 90.000,E1 15.843} C_DIS
LIN {X 0.041,Y -203.138,Z 1310.062,A 0.000,B 0.000,C 90.000,E1 11.074} C_DIS
LIN {X 0.033,Y -199.971,Z 1310.026,A 0.000,B 0.000,C 90.000,E1 4.645} C_DIS
LIN {X -0.085,Y -198.575,Z 1309.988,A 0.000,B 0.000,C 90.000,E1 357.936} C_DIS
LIN {X 0.047,Y -200.219,Z 1309.939,A 0.000,B 0.000,C 90.000,E1 348.993} C_DIS
LIN {X -0.037,Y -203.389,Z 1309.908,A 0.000,B 0.000,C 90.000,E1 343.378} C_DIS
LIN {X -0.088,Y -207.482,Z 1309.881,A 0.000,B 0.000,C 90.000,E1 338.592} C_DIS
LIN {X 0.055,Y -211.803,Z 1309.859,A 0.000,B 0.000,C 90.000,E1 334.588} C_DIS
LIN {X 0.035,Y -217.001,Z 1309.837,A 0.000,B 0.000,C 90.000,E1 330.667} C_DIS
LIN {X 0.030,Y -223.138,Z 1309.816,A 0.000,B 0.000,C 90.000,E1 326.786} C_DIS
LIN {X -0.024,Y -230.230,Z 1309.794,A 0.000,B 0.000,C 90.000,E1 322.970} C_DIS
LIN {X 0.064,Y -238.255,Z 1309.773,A 0.000,B 0.000,C 90.000,E1 319.175} C_DIS
LIN {X 0.006,Y -245.535,Z 1309.757,A 0.000,B 0.000,C 90.000,E1 316.215} C_DIS
LIN {X -0.020,Y -254.823,Z 1309.739,A 0.000,B 0.000,C 90.000,E1 312.933} C_DIS
LIN {X -0.045,Y -261.799,Z 1309.727,A 0.000,B 0.000,C 90.000,E1 310.782} C_DIS
LIN {X -0.043,Y -271.068,Z 1309.713,A 0.000,B 0.000,C 90.000,E1 308.302} C_DIS
LIN {X -0.062,Y -280.021,Z 1309.701,A 0.000,B 0.000,C 90.000,E1 306.217} C_DIS
LIN {X 0.031,Y -288.240,Z 1309.692,A 0.000,B 0.000,C 90.000,E1 304.485} C_DIS
LIN {X 0.017,Y -301.093,Z 1309.679,A 0.000,B 0.000,C 90.000,E1 302.133} C_DIS
LIN {X 0.141,Y -311.497,Z 1309.669,A 0.000,B 0.000,C 90.000,E1 300.463} C_DIS
LIN {X -0.071,Y -320.530,Z 1309.662,A 0.000,B 0.000,C 90.000,E1 299.205} C_DIS
LIN {X -0.058,Y -343.017,Z 1309.646,A 0.000,B 0.000,C 90.000,E1 296.360} C_DIS
LIN {X 0.013,Y -356.164,Z 1309.638,A 0.000,B 0.000,C 90.000,E1 294.823} C_DIS
LIN {X 0.014,Y -369.113,Z 1309.630,A 0.000,B 0.000,C 90.000,E1 293.334} C_DIS
LIN {X 0.099,Y -379.181,Z 1309.623,A 0.000,B 0.000,C 90.000,E1 292.153} C_DIS
LIN {X -0.094,Y -391.314,Z 1309.615,A 0.000,B 0.000,C 90.000,E1 290.737} C_DIS
LIN {X -0.152,Y -411.091,Z 1309.603,A 0.000,B 0.000,C 90.000,E1 288.489} C_DIS
LIN {X 0.137,Y -420.963,Z 1309.596,A 0.000,B 0.000,C 90.000,E1 287.347} C_DIS
LIN {X 0.145,Y -430.350,Z 1309.590,A 0.000,B 0.000,C 90.000,E1 286.260} C_DIS
LIN {X -0.054,Y -436.823,Z 1309.586,A 0.000,B 0.000,C 90.000,E1 285.481} C_DIS
LIN {X 0.120,Y -442.518,Z 1309.582,A 0.000,B 0.000,C 90.000,E1 284.662} C_DIS
LIN {X 0.024,Y -447.391,Z 1309.577,A 0.000,B 0.000,C 90.000,E1 283.883} C_DIS
LIN {X -0.136,Y -451.650,Z 1309.573,A 0.000,B 0.000,C 90.000,E1 283.119} C_DIS
LIN {X 0.181,Y -455.494,Z 1309.568,A 0.000,B 0.000,C 90.000,E1 282.299} C_DIS
LIN {X -0.181,Y -457.800,Z 1309.566,A 0.000,B 0.000,C 90.000,E1 281.827} C_DIS
LIN {X -0.085,Y -459.797,Z 1309.563,A 0.000,B 0.000,C 90.000,E1 281.299} C_DIS
LIN {X -0.068,Y -461.415,Z 1309.560,A 0.000,B 0.000,C 90.000,E1 280.782} C_DIS
LIN {X 0.048,Y -462.681,Z 1309.557,A 0.000,B 0.000,C 90.000,E1 280.254} C_DIS
LIN {X 0.171,Y -463.575,Z 1309.554,A 0.000,B 0.000,C 90.000,E1 279.726} C_DIS
LIN {X 0.224,Y -464.011,Z 1309.551,A 0.000,B 0.000,C 90.000,E1 279.208} C_DIS
LIN {X -0.174,Y -464.080,Z 1309.548,A 0.000,B 0.000,C 90.000,E1 278.746} C_DIS
LIN {X -0.041,Y -463.660,Z 1309.546,A 0.000,B 0.000,C 90.000,E1 278.219} C_DIS
LIN {X 0.025,Y -462.790,Z 1309.543,A 0.000,B 0.000,C 90.000,E1 277.701} C_DIS
LIN {X 0.088,Y -461.436,Z 1309.540,A 0.000,B 0.000,C 90.000,E1 277.182} C_DIS
LIN {X 0.148,Y -459.560,Z 1309.537,A 0.000,B 0.000,C 90.000,E1 276.663} C_DIS
LIN {X 0.200,Y -457.167,Z 1309.534,A 0.000,B 0.000,C 90.000,E1 276.144} C_DIS
LIN {X -0.219,Y -454.267,Z 1309.531,A 0.000,B 0.000,C 90.000,E1 275.682} C_DIS
LIN {X -0.200,Y -450.839,Z 1309.529,A 0.000,B 0.000,C 90.000,E1 275.163} C_DIS
LIN {X -0.199,Y -446.717,Z 1309.526,A 0.000,B 0.000,C 90.000,E1 274.645} C_DIS
LIN {X 0.187,Y -441.673,Z 1309.523,A 0.000,B 0.000,C 90.000,E1 274.073} C_DIS
LIN {X -0.117,Y -435.752,Z 1309.520,A 0.000,B 0.000,C 90.000,E1 273.612} C_DIS
LIN {X 0.019,Y -429.556,Z 1309.518,A 0.000,B 0.000,C 90.000,E1 273.154} C_DIS
LIN {X 0.141,Y -423.075,Z 1309.515,A 0.000,B 0.000,C 90.000,E1 272.751} C_DIS
LIN {X 0.200,Y -416.283,Z 1309.514,A 0.000,B 0.000,C 90.000,E1 272.407} C_DIS
LIN {X -0.199,Y -409.361,Z 1309.512,A 0.000,B 0.000,C 90.000,E1 272.178} C_DIS
LIN {X 0.096,Y -401.943,Z 1309.511,A 0.000,B 0.000,C 90.000,E1 271.892} C_DIS
LIN {X 0.181,Y -391.084,Z 1309.509,A 0.000,B 0.000,C 90.000,E1 271.604} C_DIS
LIN {X -0.040,Y -383.557,Z 1309.508,A 0.000,B 0.000,C 90.000,E1 271.489} C_DIS
LIN {X -0.048,Y -374.770,Z 1309.508,A 0.000,B 0.000,C 90.000,E1 271.375} C_DIS
LIN {X -0.119,Y -366.893,Z 1309.507,A 0.000,B 0.000,C 90.000,E1 271.318} C_DIS
LIN {X -0.068,Y -353.102,Z 1309.507,A 0.000,B 0.000,C 90.000,E1 271.260} C_DIS
LIN {X -0.066,Y -181.403,Z 1309.507,A 0.000,B 0.000,C 90.000,E1 271.260} C_DIS
LIN {X -0.023,Y -181.580,Z 1309.501,A 0.000,B 0.000,C 90.000,E1 270.229} C_DIS
LIN {X -0.019,Y -180.863,Z 1309.472,A 0.000,B 0.000,C 90.000,E1 265.008} C_DIS
LIN {X 0.034,Y -178.976,Z 1309.444,A 0.000,B 0.000,C 90.000,E1 259.926} C_DIS
LIN {X 0.045,Y -177.940,Z 1309.435,A 0.000,B 0.000,C 90.000,E1 258.229} C_DIS
LIN {X 0.058,Y -175.579,Z 1309.411,A 0.000,B 0.000,C 90.000,E1 253.976} C_DIS
LIN {X 0.066,Y -172.306,Z 1309.387,A 0.000,B 0.000,C 90.000,E1 249.699} C_DIS
LIN {X 0.043,Y -171.784,Z 1309.383,A 0.000,B 0.000,C 90.000,E1 248.847} C_DIS
LIN {X -0.079,Y -169.450,Z 1309.368,A 0.000,B 0.000,C 90.000,E1 246.305} C_DIS
LIN {X -0.023,Y -166.780,Z 1309.349,A 0.000,B 0.000,C 90.000,E1 242.820} C_DIS
LIN {X -0.027,Y -162.760,Z 1309.325,A 0.000,B 0.000,C 90.000,E1 238.456} C_DIS
LIN {X -0.051,Y -161.450,Z 1309.315,A 0.000,B 0.000,C 90.000,E1 236.707} C_DIS
LIN {X -0.009,Y -157.443,Z 1309.290,A 0.000,B 0.000,C 90.000,E1 232.271} C_DIS
LIN {X 0.025,Y -155.452,Z 1309.276,A 0.000,B 0.000,C 90.000,E1 229.585} C_DIS
LIN {X 0.073,Y -151.769,Z 1309.251,A 0.000,B 0.000,C 90.000,E1 225.081} C_DIS
LIN {X -0.017,Y -149.972,Z 1309.236,A 0.000,B 0.000,C 90.000,E1 222.405} C_DIS
LIN {X -0.006,Y -146.809,Z 1309.210,A 0.000,B 0.000,C 90.000,E1 217.855} C_DIS
LIN {X 0.011,Y -145.387,Z 1309.195,A 0.000,B 0.000,C 90.000,E1 215.105} C_DIS
LIN {X 0.003,Y -142.444,Z 1309.164,A 0.000,B 0.000,C 90.000,E1 209.589} C_DIS
LIN {X -0.014,Y -141.437,Z 1309.149,A 0.000,B 0.000,C 90.000,E1 206.821} C_DIS
LIN {X 0.031,Y -139.367,Z 1309.113,A 0.000,B 0.000,C 90.000,E1 200.301} C_DIS
LIN {X 0.016,Y -138.814,Z 1309.097,A 0.000,B 0.000,C 90.000,E1 197.511} C_DIS
LIN {X 0.067,Y -138.351,Z 1309.056,A 0.000,B 0.000,C 90.000,E1 190.018} C_DIS
LIN {X 0.043,Y -139.539,Z 1309.004,A 0.000,B 0.000,C 90.000,E1 180.688} C_DIS
LIN {X -0.004,Y -141.231,Z 1308.973,A 0.000,B 0.000,C 90.000,E1 175.122} C_DIS
LIN {X -0.046,Y -142.602,Z 1308.957,A 0.000,B 0.000,C 90.000,E1 172.356} C_DIS
LIN {X 0.049,Y -144.910,Z 1308.932,A 0.000,B 0.000,C 90.000,E1 167.701} C_DIS
LIN {X 0.042,Y -147.539,Z 1308.911,A 0.000,B 0.000,C 90.000,E1 164.031} C_DIS
LIN {X -0.067,Y -150.138,Z 1308.891,A 0.000,B 0.000,C 90.000,E1 160.423} C_DIS
LIN {X -0.057,Y -153.505,Z 1308.871,A 0.000,B 0.000,C 90.000,E1 156.794} C_DIS
LIN {X 0.006,Y -157.870,Z 1308.846,A 0.000,B 0.000,C 90.000,E1 152.281} C_DIS
LIN {X -0.039,Y -162.156,Z 1308.826,A 0.000,B 0.000,C 90.000,E1 148.742} C_DIS
LIN {X 0.077,Y -166.363,Z 1308.807,A 0.000,B 0.000,C 90.000,E1 145.182} C_DIS
LIN {X -0.055,Y -171.379,Z 1308.787,A 0.000,B 0.000,C 90.000,E1 141.743} C_DIS
LIN {X -0.012,Y -176.289,Z 1308.768,A 0.000,B 0.000,C 90.000,E1 138.286} C_DIS
LIN {X -0.011,Y -180.575,Z 1308.754,A 0.000,B 0.000,C 90.000,E1 135.729} C_DIS
LIN {X -0.033,Y -185.976,Z 1308.735,A 0.000,B 0.000,C 90.000,E1 132.366} C_DIS
LIN {X 0.023,Y -190.609,Z 1308.721,A 0.000,B 0.000,C 90.000,E1 129.850} C_DIS
LIN {X -0.070,Y -196.360,Z 1308.703,A 0.000,B 0.000,C 90.000,E1 126.583} C_DIS
LIN {X 0.031,Y -199.369,Z 1308.695,A 0.000,B 0.000,C 90.000,E1 125.025} C_DIS
LIN {X 0.013,Y -308.387,Z 1308.695,A 0.000,B 0.000,C 90.000,E1 125.025} C_DIS
LIN {X -0.071,Y -312.655,Z 1308.694,A 0.000,B 0.000,C 90.000,E1 124.945} C_DIS
LIN {X 0.075,Y -315.311,Z 1308.693,A 0.000,B 0.000,C 90.000,E1 124.771} C_DIS
LIN {X -0.041,Y -319.030,Z 1308.691,A 0.000,B 0.000,C 90.000,E1 124.452} C_DIS
LIN {X 0.063,Y -322.565,Z 1308.688,A 0.000,B 0.000,C 90.000,E1 123.913} C_DIS
LIN {X 0.141,Y -324.083,Z 1308.687,A 0.000,B 0.000,C 90.000,E1 123.579} C_DIS
LIN {X 0.192,Y -338.197,Z 1308.666,A 0.000,B 0.000,C 90.000,E1 119.795} C_DIS
LIN {X 0.028,Y -350.280,Z 1308.650,A 0.000,B 0.000,C 90.000,E1 117.052} C_DIS
LIN {X 0.053,Y -363.827,Z 1308.635,A 0.000,B 0.000,C 90.000,E1 114.335} C_DIS
LIN {X 0.068,Y -377.200,Z 1308.622,A 0.000,B 0.000,C 90.000,E1 111.972} C_DIS
LIN {X -0.086,Y -391.919,Z 1308.609,A 0.000,B 0.000,C 90.000,E1 109.685} C_DIS
LIN {X 0.098,Y -408.088,Z 1308.597,A 0.000,B 0.000,C 90.000,E1 107.402} C_DIS
LIN {X 0.189,Y -425.821,Z 1308.584,A 0.000,B 0.000,C 90.000,E1 105.190} C_DIS
LIN {X 0.144,Y -445.160,Z 1308.573,A 0.000,B 0.000,C 90.000,E1 103.063} C_DIS
LIN {X -0.251,Y -465.333,Z 1308.562,A 0.000,B 0.000,C 90.000,E1 101.130} C_DIS
LIN {X -0.168,Y -478.162,Z 1308.555,A 0.000,B 0.000,C 90.000,E1 99.962} C_DIS
LIN {X -0.120,Y -480.174,Z 1308.554,A 0.000,B 0.000,C 90.000,E1 99.726} C_DIS
LIN {X -0.154,Y -481.708,Z 1308.553,A 0.000,B 0.000,C 90.000,E1 99.500} C_DIS
LIN {X 0.203,Y -482.973,Z 1308.551,A 0.000,B 0.000,C 90.000,E1 99.208} C_DIS
LIN {X 0.083,Y -483.901,Z 1308.550,A 0.000,B 0.000,C 90.000,E1 98.973} C_DIS
LIN {X -0.219,Y -484.912,Z 1308.547,A 0.000,B 0.000,C 90.000,E1 98.511} C_DIS
LIN {X -0.035,Y -484.924,Z 1308.544,A 0.000,B 0.000,C 90.000,E1 97.992} C_DIS
LIN {X 0.157,Y -483.943,Z 1308.542,A 0.000,B 0.000,C 90.000,E1 97.473} C_DIS
LIN {X -0.070,Y -481.798,Z 1308.539,A 0.000,B 0.000,C 90.000,E1 97.004} C_DIS
LIN {X 0.231,Y -480.145,Z 1308.537,A 0.000,B 0.000,C 90.000,E1 96.720} C_DIS
LIN {X 0.206,Y -468.896,Z 1308.529,A 0.000,B 0.000,C 90.000,E1 95.220} C_DIS
LIN {X -0.034,Y -455.185,Z 1308.518,A 0.000,B 0.000,C 90.000,E1 93.212} C_DIS
LIN {X 0.060,Y -440.155,Z 1308.505,A 0.000,B 0.000,C 90.000,E1 90.859} C_DIS
LIN {X 0.152,Y -422.298,Z 1308.487,A 0.000,B 0.000,C 90.000,E1 87.650} C_DIS
LIN {X 0.169,Y -410.761,Z 1308.475,A 0.000,B 0.000,C 90.000,E1 85.469} C_DIS
LIN {X -0.148,Y -401.994,Z 1308.466,A 0.000,B 0.000,C 90.000,E1 83.856} C_DIS
LIN {X -0.152,Y -391.573,Z 1308.455,A 0.000,B 0.000,C 90.000,E1 81.894} C_DIS
LIN {X 0.087,Y -382.410,Z 1308.445,A 0.000,B 0.000,C 90.000,E1 80.151} C_DIS
LIN {X 0.147,Y -372.853,Z 1308.436,A 0.000,B 0.000,C 90.000,E1 78.409} C_DIS
LIN {X 0.179,Y -363.147,Z 1308.426,A 0.000,B 0.000,C 90.000,E1 76.645} C_DIS
LIN {X 0.072,Y -351.611,Z 1308.414,A 0.000,B 0.000,C 90.000,E1 74.574} C_DIS
LIN {X -0.081,Y -340.006,Z 1308.403,A 0.000,B 0.000,C 90.000,E1 72.472} C_DIS
LIN {X -0.182,Y -326.797,Z 1308.389,A 0.000,B 0.000,C 90.000,E1 70.007} C_DIS
LIN {X -0.005,Y -311.131,Z 1308.371,A 0.000,B 0.000,C 90.000,E1 66.794} C_DIS
LIN {X 0.053,Y -298.170,Z 1308.355,A 0.000,B 0.000,C 90.000,E1 63.845} C_DIS
LIN {X 0.060,Y -290.480,Z 1308.344,A 0.000,B 0.000,C 90.000,E1 61.847} C_DIS
LIN {X -0.001,Y -281.516,Z 1308.329,A 0.000,B 0.000,C 90.000,E1 59.154} C_DIS
LIN {X -0.017,Y -271.636,Z 1308.310,A 0.000,B 0.000,C 90.000,E1 55.722} C_DIS
LIN {X 0.128,Y -262.576,Z 1308.290,A 0.000,B 0.000,C 90.000,E1 52.190} C_DIS
LIN {X -0.023,Y -255.704,Z 1308.274,A 0.000,B 0.000,C 90.000,E1 49.380} C_DIS
LIN {X -0.030,Y -248.995,Z 1308.258,A 0.000,B 0.000,C 90.000,E1 46.500} C_DIS
LIN {X -0.034,Y -242.529,Z 1308.242,A 0.000,B 0.000,C 90.000,E1 43.581} C_DIS
LIN {X 0.083,Y -234.970,Z 1308.222,A 0.000,B 0.000,C 90.000,E1 39.850} C_DIS
LIN {X 0.079,Y -228.322,Z 1308.201,A 0.000,B 0.000,C 90.000,E1 36.091} C_DIS
LIN {X 0.038,Y -222.620,Z 1308.179,A 0.000,B 0.000,C 90.000,E1 32.291} C_DIS
LIN {X 0.039,Y -217.857,Z 1308.158,A 0.000,B 0.000,C 90.000,E1 28.437} C_DIS
LIN {X -0.044,Y -213.753,Z 1308.136,A 0.000,B 0.000,C 90.000,E1 24.567} C_DIS
LIN {X 0.109,Y -209.448,Z 1308.110,A 0.000,B 0.000,C 90.000,E1 19.812} C_DIS
LIN {X -0.063,Y -206.196,Z 1308.088,A 0.000,B 0.000,C 90.000,E1 15.898} C_DIS
LIN {X 0.064,Y -202.893,Z 1308.062,A 0.000,B 0.000,C 90.000,E1 11.074} C_DIS
LIN {X 0.044,Y -199.740,Z 1308.026,A 0.000,B 0.000,C 90.000,E1 4.645} C_DIS
LIN {X -0.064,Y -198.447,Z 1307.993,A 0.000,B 0.000,C 90.000,E1 358.740} C_DIS
LIN {X 0.034,Y -200.114,Z 1307.939,A 0.000,B 0.000,C 90.000,E1 348.993} C_DIS
LIN {X -0.055,Y -203.365,Z 1307.908,A 0.000,B 0.000,C 90.000,E1 343.378} C_DIS
LIN {X -0.106,Y -207.512,Z 1307.881,A 0.000,B 0.000,C 90.000,E1 338.592} C_DIS
LIN {X 0.037,Y -211.874,Z 1307.859,A 0.000,B 0.000,C 90.000,E1 334.588} C_DIS
LIN {X 0.019,Y -217.078,Z 1307.837,A 0.000,B 0.000,C 90.000,E1 330.667} C_DIS
LIN {X 0.017,Y -223.216,Z 1307.816,A 0.000,B 0.000,C 90.000,E1 326.786} C_DIS
LIN {X -0.034,Y -230.318,Z 1307.794,A 0.000,B 0.000,C 90.000,E1 322.970} C_DIS
LIN {X 0.055,Y -238.320,Z 1307.773,A 0.000,B 0.000,C 90.000,E1 319.175} C_DIS
LIN {X -0.002,Y -245.604,Z 1307.757,A 0.000,B 0.000,C 90.000,E1 316.215} C_DIS
LIN {X -0.026,Y -254.875,Z 1307.739,A 0.000,B 0.000,C 90.000,E1 312.933} C_DIS
LIN {X -0.050,Y -261.826,Z 1307.727,A 0.000,B 0.000,C 90.000,E1 310.782} C_DIS
LIN {X 0.033,Y -272.515,Z 1307.711,A 0.000,B 0.000,C 90.000,E1 307.935} C_DIS
LIN {X -0.013,Y -283.234,Z 1307.697,A 0.000,B 0.000,C 90.000,E1 305.518} C_DIS
LIN {X 0.136,Y -291.817,Z 1307.688,A 0.000,B 0.000,C 90.000,E1 303.785} C_DIS
LIN {X 0.027,Y -303.118,Z 1307.677,A 0.000,B 0.000,C 90.000,E1 301.799} C_DIS
LIN {X -0.195,Y -315.944,Z 1307.666,A 0.000,B 0.000,C 90.000,E1 299.873} C_DIS
LIN {X 0.139,Y -330.234,Z 1307.655,A 0.000,B 0.000,C 90.000,E1 297.897} C_DIS
LIN {X -0.091,Y -353.447,Z 1307.640,A 0.000,B 0.000,C 90.000,E1 295.155} C_DIS
LIN {X 0.028,Y -366.391,Z 1307.631,A 0.000,B 0.000,C 90.000,E1 293.643} C_DIS
LIN {X 0.132,Y -379.106,Z 1307.623,A 0.000,B 0.000,C 90.000,E1 292.153} C_DIS
LIN {X -0.061,Y -391.261,Z 1307.615,A 0.000,B 0.000,C 90.000,E1 290.737} C_DIS
LIN {X -0.120,Y -411.046,Z 1307.603,A 0.000,B 0.000,C 90.000,E1 288.489} C_DIS
LIN {X 0.016,Y -423.347,Z 1307.595,A 0.000,B 0.000,C 90.000,E1 287.094} C_DIS
LIN {X -0.077,Y -432.552,Z 1307.589,A 0.000,B 0.000,C 90.000,E1 286.024} C_DIS
LIN {X 0.171,Y -438.833,Z 1307.584,A 0.000,B 0.000,C 90.000,E1 285.190} C_DIS
LIN {X 0.044,Y -444.207,Z 1307.580,A 0.000,B 0.000,C 90.000,E1 284.411} C_DIS
LIN {X -0.146,Y -448.864,Z 1307.576,A 0.000,B 0.000,C 90.000,E1 283.647} C_DIS
LIN {X -0.043,Y -454.222,Z 1307.570,A 0.000,B 0.000,C 90.000,E1 282.591} C_DIS
LIN {X -0.149,Y -457.760,Z 1307.566,A 0.000,B 0.000,C 90.000,E1 281.827} C_DIS
LIN {X -0.053,Y -459.758,Z 1307.563,A 0.000,B 0.000,C 90.000,E1 281.299} C_DIS
LIN {X -0.037,Y -461.393,Z 1307.560,A 0.000,B 0.000,C 90.000,E1 280.782} C_DIS
LIN {X 0.080,Y -462.707,Z 1307.557,A 0.000,B 0.000,C 90.000,E1 280.254} C_DIS
LIN {X 0.203,Y -463.622,Z 1307.554,A 0.000,B 0.000,C 90.000,E1 279.726} C_DIS
LIN {X -0.202,Y -464.159,Z 1307.551,A 0.000,B 0.000,C 90.000,E1 279.265} C_DIS
LIN {X -0.141,Y -464.210,Z 1307.548,A 0.000,B 0.000,C 90.000,E1 278.746} C_DIS
LIN {X -0.008,Y -463.881,Z 1307.546,A 0.000,B 0.000,C 90.000,E1 278.219} C_DIS
LIN {X 0.058,Y -463.015,Z 1307.543,A 0.000,B 0.000,C 90.000,E1 277.701} C_DIS
LIN {X 0.123,Y -461.723,Z 1307.540,A 0.000,B 0.000,C 90.000,E1 277.182} C_DIS
LIN {X 0.184,Y -459.866,Z 1307.537,A 0.000,B 0.000,C 90.000,E1 276.663} C_DIS
LIN {X 0.051,Y -456.157,Z 1307.533,A 0.000,B 0.000,C 90.000,E1 275.910} C_DIS
LIN {X 0.077,Y -453.079,Z 1307.530,A 0.000,B 0.000,C 90.000,E1 275.391} C_DIS
LIN {X 0.047,Y -449.448,Z 1307.527,A 0.000,B 0.000,C 90.000,E1 274.878} C_DIS
LIN {X 0.038,Y -444.939,Z 1307.524,A 0.000,B 0.000,C 90.000,E1 274.359} C_DIS
LIN {X 0.073,Y -439.502,Z 1307.521,A 0.000,B 0.000,C 90.000,E1 273.841} C_DIS
LIN {X -0.069,Y -433.480,Z 1307.519,A 0.000,B 0.000,C 90.000,E1 273.383} C_DIS
LIN {X -0.188,Y -427.167,Z 1307.516,A 0.000,B 0.000,C 90.000,E1 272.980} C_DIS
LIN {X 0.063,Y -420.518,Z 1307.514,A 0.000,B 0.000,C 90.000,E1 272.579} C_DIS
LIN {X -0.149,Y -413.597,Z 1307.513,A 0.000,B 0.000,C 90.000,E1 272.293} C_DIS
LIN {X -0.007,Y -406.453,Z 1307.511,A 0.000,B 0.000,C 90.000,E1 272.007} C_DIS
LIN {X 0.080,Y -399.064,Z 1307.510,A 0.000,B 0.000,C 90.000,E1 271.776} C_DIS
LIN {X -0.119,Y -387.944,Z 1307.509,A 0.000,B 0.000,C 90.000,E1 271.547} C_DIS
LIN {X 0.129,Y -379.552,Z 1307.508,A 0.000,B 0.000,C 90.000,E1 271.375} C_DIS
LIN {X -0.149,Y -370.275,Z 1307.507,A 0.000,B 0.000,C 90.000,E1 271.318} C_DIS
LIN {X 0.138,Y -354.401,Z 1307.507,A 0.000,B 0.000,C 90.000,E1 271.203} C_DIS
LIN {X 0.039,Y -181.409,Z 1307.507,A 0.000,B 0.000,C 90.000,E1 271.203} C_DIS
LIN {X 0.083,Y -181.580,Z 1307.501,A 0.000,B 0.000,C 90.000,E1 270.172} C_DIS
LIN {X 0.087,Y -180.857,Z 1307.472,A 0.000,B 0.000,C 90.000,E1 264.951} C_DIS
LIN {X -0.039,Y -178.968,Z 1307.444,A 0.000,B 0.000,C 90.000,E1 259.926} C_DIS
LIN {X -0.029,Y -177.923,Z 1307.435,A 0.000,B 0.000,C 90.000,E1 258.229} C_DIS
LIN {X -0.015,Y -175.560,Z 1307.411,A 0.000,B 0.000,C 90.000,E1 253.976} C_DIS
LIN {X -0.007,Y -172.290,Z 1307.387,A 0.000,B 0.000,C 90.000,E1 249.699} C_DIS
LIN {X -0.029,Y -171.769,Z 1307.382,A 0.000,B 0.000,C 90.000,E1 248.847} C_DIS
LIN {X -0.037,Y -168.010,Z 1307.359,A 0.000,B 0.000,C 90.000,E1 244.537} C_DIS
LIN {X -0.018,Y -166.761,Z 1307.349,A 0.000,B 0.000,C 90.000,E1 242.794} C_DIS
LIN {X 0.041,Y -162.740,Z 1307.325,A 0.000,B 0.000,C 90.000,E1 238.408} C_DIS
LIN {X 0.103,Y -161.431,Z 1307.315,A 0.000,B 0.000,C 90.000,E1 236.628} C_DIS
LIN {X -0.078,Y -157.424,Z 1307.290,A 0.000,B 0.000,C 90.000,E1 232.271} C_DIS
LIN {X 0.075,Y -155.427,Z 1307.275,A 0.000,B 0.000,C 90.000,E1 229.542} C_DIS
LIN {X 0.006,Y -151.752,Z 1307.250,A 0.000,B 0.000,C 90.000,E1 225.081} C_DIS
LIN {X 0.017,Y -149.952,Z 1307.235,A 0.000,B 0.000,C 90.000,E1 222.366} C_DIS
LIN {X 0.045,Y -146.795,Z 1307.210,A 0.000,B 0.000,C 90.000,E1 217.810} C_DIS
LIN {X -0.055,Y -145.370,Z 1307.195,A 0.000,B 0.000,C 90.000,E1 215.105} C_DIS
LIN {X 0.062,Y -142.434,Z 1307.164,A 0.000,B 0.000,C 90.000,E1 209.539} C_DIS
LIN {X -0.015,Y -141.424,Z 1307.149,A 0.000,B 0.000,C 90.000,E1 206.796} C_DIS
LIN {X -0.033,Y -139.363,Z 1307.113,A 0.000,B 0.000,C 90.000,E1 200.301} C_DIS
LIN {X -0.047,Y -138.807,Z 1307.097,A 0.000,B 0.000,C 90.000,E1 197.511} C_DIS
LIN {X 0.003,Y -138.350,Z 1307.056,A 0.000,B 0.000,C 90.000,E1 190.018} C_DIS
LIN {X -0.021,Y -139.543,Z 1307.004,A 0.000,B 0.000,C 90.000,E1 180.688} C_DIS
LIN {X 0.073,Y -141.242,Z 1306.973,A 0.000,B 0.000,C 90.000,E1 175.065} C_DIS
LIN {X 0.031,Y -142.612,Z 1306.957,A 0.000,B 0.000,C 90.000,E1 172.299} C_DIS
LIN {X -0.016,Y -144.927,Z 1306.932,A 0.000,B 0.000,C 90.000,E1 167.701} C_DIS
LIN {X -0.024,Y -147.555,Z 1306.911,A 0.000,B 0.000,C 90.000,E1 164.031} C_DIS
LIN {X 0.007,Y -150.159,Z 1306.891,A 0.000,B 0.000,C 90.000,E1 160.369} C_DIS
LIN {X 0.017,Y -153.532,Z 1306.871,A 0.000,B 0.000,C 90.000,E1 156.741} C_DIS
LIN {X 0.070,Y -156.949,Z 1306.851,A 0.000,B 0.000,C 90.000,E1 153.127} C_DIS
LIN {X 0.005,Y -161.054,Z 1306.831,A 0.000,B 0.000,C 90.000,E1 149.587} C_DIS
LIN {X 0.091,Y -163.163,Z 1306.821,A 0.000,B 0.000,C 90.000,E1 147.788} C_DIS
LIN {X -0.039,Y -167.581,Z 1306.802,A 0.000,B 0.000,C 90.000,E1 144.322} C_DIS
LIN {X 0.007,Y -171.411,Z 1306.787,A 0.000,B 0.000,C 90.000,E1 141.698} C_DIS
LIN {X 0.046,Y -176.327,Z 1306.768,A 0.000,B 0.000,C 90.000,E1 138.243} C_DIS
LIN {X -0.086,Y -180.616,Z 1306.754,A 0.000,B 0.000,C 90.000,E1 135.729} C_DIS
LIN {X 0.028,Y -186.017,Z 1306.735,A 0.000,B 0.000,C 90.000,E1 132.324} C_DIS
LIN {X -0.054,Y -190.652,Z 1306.721,A 0.000,B 0.000,C 90.000,E1 129.850} C_DIS
LIN {X 0.009,Y -196.403,Z 1306.703,A 0.000,B 0.000,C 90.000,E1 126.537} C_DIS
LIN {X -0.023,Y -199.401,Z 1306.695,A 0.000,B 0.000,C 90.000,E1 125.025} C_DIS
LIN {X -0.071,Y -309.129,Z 1306.694,A 0.000,B 0.000,C 90.000,E1 125.025} C_DIS
LIN {X 0.061,Y -312.938,Z 1306.694,A 0.000,B 0.000,C 90.000,E1 124.898} C_DIS
LIN {X -0.088,Y -316.024,Z 1306.693,A 0.000,B 0.000,C 90.000,E1 124.739} C_DIS
LIN {X 0.167,Y -319.696,Z 1306.691,A 0.000,B 0.000,C 90.000,E1 124.326} C_DIS
LIN {X 0.059,Y -323.179,Z 1306.688,A 0.000,B 0.000,C 90.000,E1 123.785} C_DIS
LIN {X -0.130,Y -324.566,Z 1306.686,A 0.000,B 0.000,C 90.000,E1 123.499} C_DIS
LIN {X -0.057,Y -336.173,Z 1306.668,A 0.000,B 0.000,C 90.000,E1 120.335} C_DIS
LIN {X 0.192,Y -348.006,Z 1306.653,A 0.000,B 0.000,C 90.000,E1 117.513} C_DIS
LIN {X -0.014,Y -361.285,Z 1306.638,A 0.000,B 0.000,C 90.000,E1 114.823} C_DIS
LIN {X -0.074,Y -374.399,Z 1306.625,A 0.000,B 0.000,C 90.000,E1 112.461} C_DIS
LIN {X 0.062,Y -388.841,Z 1306.612,A 0.000,B 0.000,C 90.000,E1 110.120} C_DIS
LIN {X -0.081,Y -404.712,Z 1306.599,A 0.000,B 0.000,C 90.000,E1 107.873} C_DIS
LIN {X -0.089,Y -422.122,Z 1306.587,A 0.000,B 0.000,C 90.000,E1 105.662} C_DIS
LIN {X 0.142,Y -441.174,Z 1306.575,A 0.000,B 0.000,C 90.000,E1 103.480} C_DIS
LIN {X 0.024,Y -461.234,Z 1306.564,A 0.000,B 0.000,C 90.000,E1 101.478} C_DIS
LIN {X 0.024,Y -476.638,Z 1306.556,A 0.000,B 0.000,C 90.000,E1 100.074} C_DIS
LIN {X 0.016,Y -478.972,Z 1306.555,A 0.000,B 0.000,C 90.000,E1 99.849} C_DIS
LIN {X -0.032,Y -480.832,Z 1306.553,A 0.000,B 0.000,C 90.000,E1 99.613} C_DIS
LIN {X -0.082,Y -482.241,Z 1306.552,A 0.000,B 0.000,C 90.000,E1 99.378} C_DIS
LIN {X 0.081,Y -484.110,Z 1306.549,A 0.000,B 0.000,C 90.000,E1 98.859} C_DIS
LIN {X -0.225,Y -484.867,Z 1306.547,A 0.000,B 0.000,C 90.000,E1 98.398} C_DIS
LIN {X 0.029,Y -484.639,Z 1306.544,A 0.000,B 0.000,C 90.000,E1 97.871} C_DIS
LIN {X 0.217,Y -483.394,Z 1306.541,A 0.000,B 0.000,C 90.000,E1 97.352} C_DIS
LIN {X 0.042,Y -482.332,Z 1306.540,A 0.000,B 0.000,C 90.000,E1 97.125} C_DIS
LIN {X -0.073,Y -480.903,Z 1306.538,A 0.000,B 0.000,C 90.000,E1 96.891} C_DIS
LIN {X 0.182,Y -467.906,Z 1306.528,A 0.000,B 0.000,C 90.000,E1 95.106} C_DIS
LIN {X -0.052,Y -454.188,Z 1306.517,A 0.000,B 0.000,C 90.000,E1 93.094} C_DIS
LIN {X -0.004,Y -439.213,Z 1306.504,A 0.000,B 0.000,C 90.000,E1 90.745} C_DIS
LIN {X -0.065,Y -422.859,Z 1306.488,A 0.000,B 0.000,C 90.000,E1 87.822} C_DIS
LIN {X -0.027,Y -411.325,Z 1306.476,A 0.000,B 0.000,C 90.000,E1 85.641} C_DIS
LIN {X -0.018,Y -404.026,Z 1306.468,A 0.000,B 0.000,C 90.000,E1 84.261} C_DIS
LIN {X 0.015,Y -393.667,Z 1306.457,A 0.000,B 0.000,C 90.000,E1 82.299} C_DIS
LIN {X -0.155,Y -384.611,Z 1306.448,A 0.000,B 0.000,C 90.000,E1 80.622} C_DIS
LIN {X 0.020,Y -375.106,Z 1306.438,A 0.000,B 0.000,C 90.000,E1 78.870} C_DIS
LIN {X 0.021,Y -365.460,Z 1306.428,A 0.000,B 0.000,C 90.000,E1 77.117} C_DIS
LIN {X 0.012,Y -355.605,Z 1306.419,A 0.000,B 0.000,C 90.000,E1 75.338} C_DIS
LIN {X -0.166,Y -345.679,Z 1306.408,A 0.000,B 0.000,C 90.000,E1 73.559} C_DIS
LIN {X 0.001,Y -335.721,Z 1306.398,A 0.000,B 0.000,C 90.000,E1 71.692} C_DIS
LIN {X 0.103,Y -319.514,Z 1306.381,A 0.000,B 0.000,C 90.000,E1 68.539} C_DIS
LIN {X -0.084,Y -302.973,Z 1306.361,A 0.000,B 0.000,C 90.000,E1 65.025} C_DIS
LIN {X 0.019,Y -293.502,Z 1306.348,A 0.000,B 0.000,C 90.000,E1 62.692} C_DIS
LIN {X 0.058,Y -285.276,Z 1306.335,A 0.000,B 0.000,C 90.000,E1 60.333} C_DIS
LIN {X 0.174,Y -276.931,Z 1306.320,A 0.000,B 0.000,C 90.000,E1 57.582} C_DIS
LIN {X 0.014,Y -267.440,Z 1306.301,A 0.000,B 0.000,C 90.000,E1 54.149} C_DIS
LIN {X -0.077,Y -258.646,Z 1306.281,A 0.000,B 0.000,C 90.000,E1 50.642} C_DIS
LIN {X 0.012,Y -251.851,Z 1306.265,A 0.000,B 0.000,C 90.000,E1 47.757} C_DIS
LIN {X 0.066,Y -243.675,Z 1306.245,A 0.000,B 0.000,C 90.000,E1 44.109} C_DIS
LIN {X -0.120,Y -235.952,Z 1306.225,A 0.000,B 0.000,C 90.000,E1 40.458} C_DIS
LIN {X 0.054,Y -229.166,Z 1306.204,A 0.000,B 0.000,C 90.000,E1 36.664} C_DIS
LIN {X -0.022,Y -223.304,Z 1306.183,A 0.000,B 0.000,C 90.000,E1 32.880} C_DIS
LIN {X -0.005,Y -218.406,Z 1306.161,A 0.000,B 0.000,C 90.000,E1 29.027} C_DIS
LIN {X 0.080,Y -213.394,Z 1306.135,A 0.000,B 0.000,C 90.000,E1 24.335} C_DIS
LIN {X -0.002,Y -209.743,Z 1306.114,A 0.000,B 0.000,C 90.000,E1 20.429} C_DIS
LIN {X -0.096,Y -206.404,Z 1306.092,A 0.000,B 0.000,C 90.000,E1 16.496} C_DIS
LIN {X 0.015,Y -203.519,Z 1306.069,A 0.000,B 0.000,C 90.000,E1 12.479} C_DIS
LIN {X 0.101,Y -200.384,Z 1306.038,A 0.000,B 0.000,C 90.000,E1 6.834} C_DIS
LIN {X 0.000,Y -198.394,Z 1306.000,A 0.000,B 0.000,C 90.000,E1 360.000} C_DIS
LIN {X 0.017,Y -199.659,Z 1305.943,A 0.000,B 0.000,C 90.000,E1 349.803} C_DIS
LIN {X 0.013,Y -202.763,Z 1305.912,A 0.000,B 0.000,C 90.000,E1 344.157} C_DIS
LIN {X 0.065,Y -206.767,Z 1305.885,A 0.000,B 0.000,C 90.000,E1 339.337} C_DIS
LIN {X 0.098,Y -210.981,Z 1305.863,A 0.000,B 0.000,C 90.000,E1 335.357} C_DIS
LIN {X 0.054,Y -216.031,Z 1305.841,A 0.000,B 0.000,C 90.000,E1 331.435} C_DIS
LIN {X -0.086,Y -221.986,Z 1305.820,A 0.000,B 0.000,C 90.000,E1 327.582} C_DIS
LIN {X 0.065,Y -228.918,Z 1305.798,A 0.000,B 0.000,C 90.000,E1 323.703} C_DIS
LIN {X 0.112,Y -236.696,Z 1305.777,A 0.000,B 0.000,C 90.000,E1 319.908} C_DIS
LIN {X 0.033,Y -243.755,Z 1305.761,A 0.000,B 0.000,C 90.000,E1 316.944} C_DIS
LIN {X 0.122,Y -252.781,Z 1305.743,A 0.000,B 0.000,C 90.000,E1 313.623} C_DIS
LIN {X -0.100,Y -260.621,Z 1305.729,A 0.000,B 0.000,C 90.000,E1 311.148} C_DIS
LIN {X -0.054,Y -271.135,Z 1305.713,A 0.000,B 0.000,C 90.000,E1 308.302} C_DIS
LIN {X -0.129,Y -281.620,Z 1305.699,A 0.000,B 0.000,C 90.000,E1 305.884} C_DIS
LIN {X 0.151,Y -290.063,Z 1305.690,A 0.000,B 0.000,C 90.000,E1 304.119} C_DIS
LIN {X 0.007,Y -301.171,Z 1305.678,A 0.000,B 0.000,C 90.000,E1 302.133} C_DIS
LIN {X 0.064,Y -307.291,Z 1305.673,A 0.000,B 0.000,C 90.000,E1 301.131} C_DIS
LIN {X -0.147,Y -318.273,Z 1305.664,A 0.000,B 0.000,C 90.000,E1 299.539} C_DIS
LIN {X 0.109,Y -332.733,Z 1305.653,A 0.000,B 0.000,C 90.000,E1 297.590} C_DIS
LIN {X -0.101,Y -353.442,Z 1305.640,A 0.000,B 0.000,C 90.000,E1 295.155} C_DIS
LIN {X -0.009,Y -366.436,Z 1305.631,A 0.000,B 0.000,C 90.000,E1 293.643} C_DIS
LIN {X 0.091,Y -379.146,Z 1305.623,A 0.000,B 0.000,C 90.000,E1 292.153} C_DIS
LIN {X -0.104,Y -391.300,Z 1305.615,A 0.000,B 0.000,C 90.000,E1 290.737} C_DIS
LIN {X -0.033,Y -411.084,Z 1305.603,A 0.000,B 0.000,C 90.000,E1 288.471} C_DIS
LIN {X -0.028,Y -423.382,Z 1305.595,A 0.000,B 0.000,C 90.000,E1 287.094} C_DIS
LIN {X -0.121,Y -432.644,Z 1305.589,A 0.000,B 0.000,C 90.000,E1 286.024} C_DIS
LIN {X 0.126,Y -438.881,Z 1305.584,A 0.000,B 0.000,C 90.000,E1 285.190} C_DIS
LIN {X -0.001,Y -444.273,Z 1305.580,A 0.000,B 0.000,C 90.000,E1 284.411} C_DIS
LIN {X -0.190,Y -448.925,Z 1305.576,A 0.000,B 0.000,C 90.000,E1 283.647} C_DIS
LIN {X -0.089,Y -454.274,Z 1305.570,A 0.000,B 0.000,C 90.000,E1 282.591} C_DIS
LIN {X -0.194,Y -457.784,Z 1305.566,A 0.000,B 0.000,C 90.000,E1 281.827} C_DIS
LIN {X -0.097,Y -459.776,Z 1305.563,A 0.000,B 0.000,C 90.000,E1 281.299} C_DIS
LIN {X -0.082,Y -461.441,Z 1305.560,A 0.000,B 0.000,C 90.000,E1 280.782} C_DIS
LIN {X 0.035,Y -462.769,Z 1305.557,A 0.000,B 0.000,C 90.000,E1 280.254} C_DIS
LIN {X 0.159,Y -463.723,Z 1305.554,A 0.000,B 0.000,C 90.000,E1 279.726} C_DIS
LIN {X 0.212,Y -464.271,Z 1305.551,A 0.000,B 0.000,C 90.000,E1 279.208} C_DIS
LIN {X -0.185,Y -464.393,Z 1305.548,A 0.000,B 0.000,C 90.000,E1 278.746} C_DIS
LIN {X -0.051,Y -464.051,Z 1305.546,A 0.000,B 0.000,C 90.000,E1 278.219} C_DIS
LIN {X 0.015,Y -463.223,Z 1305.543,A 0.000,B 0.000,C 90.000,E1 277.701} C_DIS
LIN {X 0.083,Y -461.905,Z 1305.540,A 0.000,B 0.000,C 90.000,E1 277.182} C_DIS
LIN {X -0.031,Y -459.022,Z 1305.536,A 0.000,B 0.000,C 90.000,E1 276.429} C_DIS
LIN {X -0.217,Y -455.053,Z 1305.531,A 0.000,B 0.000,C 90.000,E1 275.682} C_DIS
LIN {X -0.194,Y -451.743,Z 1305.529,A 0.000,B 0.000,C 90.000,E1 275.163} C_DIS
LIN {X -0.188,Y -447.755,Z 1305.526,A 0.000,B 0.000,C 90.000,E1 274.645} C_DIS
LIN {X 0.204,Y -442.900,Z 1305.523,A 0.000,B 0.000,C 90.000,E1 274.073} C_DIS
LIN {X -0.202,Y -436.974,Z 1305.520,A 0.000,B 0.000,C 90.000,E1 273.612} C_DIS
LIN {X -0.127,Y -430.830,Z 1305.517,A 0.000,B 0.000,C 90.000,E1 273.151} C_DIS
LIN {X -0.098,Y -424.232,Z 1305.515,A 0.000,B 0.000,C 90.000,E1 272.751} C_DIS
LIN {X -0.047,Y -417.553,Z 1305.513,A 0.000,B 0.000,C 90.000,E1 272.407} C_DIS
LIN {X -0.052,Y -410.702,Z 1305.512,A 0.000,B 0.000,C 90.000,E1 272.121} C_DIS
LIN {X -0.170,Y -403.393,Z 1305.510,A 0.000,B 0.000,C 90.000,E1 271.892} C_DIS
LIN {X -0.089,Y -392.587,Z 1305.509,A 0.000,B 0.000,C 90.000,E1 271.604} C_DIS
LIN {X 0.086,Y -385.122,Z 1305.508,A 0.000,B 0.000,C 90.000,E1 271.432} C_DIS
LIN {X 0.065,Y -376.679,Z 1305.507,A 0.000,B 0.000,C 90.000,E1 271.318} C_DIS
LIN {X -0.165,Y -365.672,Z 1305.507,A 0.000,B 0.000,C 90.000,E1 271.260} C_DIS
LIN {X -0.057,Y -351.854,Z 1305.507,A 0.000,B 0.000,C 90.000,E1 271.203} C_DIS
LIN {X -0.062,Y -181.416,Z 1305.507,A 0.000,B 0.000,C 90.000,E1 271.203} C_DIS
LIN {X 0.077,Y -181.581,Z 1305.502,A 0.000,B 0.000,C 90.000,E1 270.286} C_DIS
LIN {X 0.052,Y -180.901,Z 1305.474,A 0.000,B 0.000,C 90.000,E1 265.241} C_DIS
LIN {X 0.001,Y -180.225,Z 1305.464,A 0.000,B 0.000,C 90.000,E1 263.571} C_DIS
LIN {X -0.046,Y -179.039,Z 1305.446,A 0.000,B 0.000,C 90.000,E1 260.208} C_DIS
LIN {X 0.017,Y -178.706,Z 1305.441,A 0.000,B 0.000,C 90.000,E1 259.342} C_DIS
LIN {X -0.042,Y -175.755,Z 1305.412,A 0.000,B 0.000,C 90.000,E1 254.267} C_DIS
LIN {X -0.039,Y -171.938,Z 1305.384,A 0.000,B 0.000,C 90.000,E1 249.135} C_DIS
LIN {X -0.063,Y -171.319,Z 1305.379,A 0.000,B 0.000,C 90.000,E1 248.284} C_DIS
LIN {X -0.010,Y -167.578,Z 1305.355,A 0.000,B 0.000,C 90.000,E1 243.948} C_DIS
LIN {X -0.071,Y -166.210,Z 1305.346,A 0.000,B 0.000,C 90.000,E1 242.231} C_DIS
LIN {X -0.081,Y -162.974,Z 1305.326,A 0.000,B 0.000,C 90.000,E1 238.742} C_DIS
LIN {X -0.034,Y -160.888,Z 1305.312,A 0.000,B 0.000,C 90.000,E1 236.087} C_DIS
LIN {X -0.056,Y -157.657,Z 1305.292,A 0.000,B 0.000,C 90.000,E1 232.557} C_DIS
LIN {X 0.002,Y -155.695,Z 1305.277,A 0.000,B 0.000,C 90.000,E1 229.865} C_DIS
LIN {X -0.062,Y -151.959,Z 1305.252,A 0.000,B 0.000,C 90.000,E1 225.405} C_DIS
LIN {X -0.045,Y -150.200,Z 1305.237,A 0.000,B 0.000,C 90.000,E1 222.690} C_DIS
LIN {X 0.086,Y -146.969,Z 1305.212,A 0.000,B 0.000,C 90.000,E1 218.096} C_DIS
LIN {X -0.011,Y -145.556,Z 1305.197,A 0.000,B 0.000,C 90.000,E1 215.391} C_DIS
LIN {X -0.011,Y -142.948,Z 1305.171,A 0.000,B 0.000,C 90.000,E1 210.797} C_DIS
LIN {X 0.046,Y -141.574,Z 1305.151,A 0.000,B 0.000,C 90.000,E1 207.078} C_DIS
LIN {X -0.033,Y -139.414,Z 1305.114,A 0.000,B 0.000,C 90.000,E1 200.610} C_DIS
LIN {X 0.020,Y -139.137,Z 1305.104,A 0.000,B 0.000,C 90.000,E1 198.725} C_DIS
LIN {X 0.046,Y -138.349,Z 1305.057,A 0.000,B 0.000,C 90.000,E1 190.310} C_DIS
LIN {X 0.034,Y -139.494,Z 1305.005,A 0.000,B 0.000,C 90.000,E1 180.974} C_DIS
LIN {X -0.025,Y -141.108,Z 1304.974,A 0.000,B 0.000,C 90.000,E1 175.412} C_DIS
LIN {X -0.071,Y -142.487,Z 1304.959,A 0.000,B 0.000,C 90.000,E1 172.648} C_DIS
LIN {X 0.017,Y -144.738,Z 1304.933,A 0.000,B 0.000,C 90.000,E1 167.993} C_DIS
LIN {X -0.033,Y -147.344,Z 1304.913,A 0.000,B 0.000,C 90.000,E1 164.338} C_DIS
LIN {X 0.032,Y -150.668,Z 1304.888,A 0.000,B 0.000,C 90.000,E1 159.752} C_DIS
LIN {X -0.088,Y -154.147,Z 1304.867,A 0.000,B 0.000,C 90.000,E1 156.177} C_DIS
LIN {X 0.047,Y -157.577,Z 1304.848,A 0.000,B 0.000,C 90.000,E1 152.538} C_DIS
LIN {X -0.001,Y -161.824,Z 1304.828,A 0.000,B 0.000,C 90.000,E1 148.997} C_DIS
LIN {X 0.017,Y -166.014,Z 1304.808,A 0.000,B 0.000,C 90.000,E1 145.468} C_DIS
LIN {X 0.009,Y -171.015,Z 1304.789,A 0.000,B 0.000,C 90.000,E1 141.984} C_DIS
LIN {X 0.041,Y -175.885,Z 1304.770,A 0.000,B 0.000,C 90.000,E1 138.528} C_DIS
LIN {X -0.083,Y -181.489,Z 1304.751,A 0.000,B 0.000,C 90.000,E1 135.162} C_DIS
LIN {X 0.053,Y -187.004,Z 1304.732,A 0.000,B 0.000,C 90.000,E1 131.757} C_DIS
LIN {X 0.055,Y -190.122,Z 1304.723,A 0.000,B 0.000,C 90.000,E1 130.092} C_DIS
LIN {X 0.074,Y -195.894,Z 1304.704,A 0.000,B 0.000,C 90.000,E1 126.790} C_DIS
LIN {X -0.040,Y -199.411,Z 1304.695,A 0.000,B 0.000,C 90.000,E1 125.025} C_DIS
LIN {X -0.111,Y -308.449,Z 1304.694,A 0.000,B 0.000,C 90.000,E1 125.025} C_DIS
LIN {X 0.043,Y -310.161,Z 1304.694,A 0.000,B 0.000,C 90.000,E1 124.978} C_DIS
LIN {X 0.070,Y -314.253,Z 1304.693,A 0.000,B 0.000,C 90.000,E1 124.818} C_DIS
LIN {X -0.084,Y -316.477,Z 1304.693,A 0.000,B 0.000,C 90.000,E1 124.692} C_DIS
LIN {X 0.049,Y -319.527,Z 1304.691,A 0.000,B 0.000,C 90.000,E1 124.358} C_DIS
LIN {X 0.088,Y -323.114,Z 1304.688,A 0.000,B 0.000,C 90.000,E1 123.785} C_DIS
LIN {X -0.102,Y -324.520,Z 1304.686,A 0.000,B 0.000,C 90.000,E1 123.499} C_DIS
LIN {X -0.029,Y -336.133,Z 1304.668,A 0.000,B 0.000,C 90.000,E1 120.335} C_DIS
LIN {X -0.089,Y -347.963,Z 1304.653,A 0.000,B 0.000,C 90.000,E1 117.564} C_DIS
LIN {X 0.014,Y -361.238,Z 1304.638,A 0.000,B 0.000,C 90.000,E1 114.823} C_DIS
LIN {X -0.046,Y -374.350,Z 1304.625,A 0.000,B 0.000,C 90.000,E1 112.461} C_DIS
LIN {X 0.091,Y -388.790,Z 1304.612,A 0.000,B 0.000,C 90.000,E1 110.120} C_DIS
LIN {X -0.054,Y -404.657,Z 1304.599,A 0.000,B 0.000,C 90.000,E1 107.873} C_DIS
LIN {X -0.062,Y -422.065,Z 1304.587,A 0.000,B 0.000,C 90.000,E1 105.662} C_DIS
LIN {X 0.169,Y -441.114,Z 1304.575,A 0.000,B 0.000,C 90.000,E1 103.480} C_DIS
LIN {X 0.049,Y -461.172,Z 1304.564,A 0.000,B 0.000,C 90.000,E1 101.478} C_DIS
LIN {X 0.047,Y -476.575,Z 1304.556,A 0.000,B 0.000,C 90.000,E1 100.074} C_DIS
LIN {X 0.039,Y -478.897,Z 1304.555,A 0.000,B 0.000,C 90.000,E1 99.849} C_DIS
LIN {X -0.016,Y -480.752,Z 1304.553,A 0.000,B 0.000,C 90.000,E1 99.613} C_DIS
LIN {X -0.074,Y -482.154,Z 1304.552,A 0.000,B 0.000,C 90.000,E1 99.378} C_DIS
LIN {X 0.088,Y -484.006,Z 1304.549,A 0.000,B 0.000,C 90.000,E1 98.859} C_DIS
LIN {X -0.217,Y -484.747,Z 1304.547,A 0.000,B 0.000,C 90.000,E1 98.398} C_DIS
LIN {X 0.035,Y -484.506,Z 1304.544,A 0.000,B 0.000,C 90.000,E1 97.871} C_DIS
LIN {X 0.224,Y -483.247,Z 1304.541,A 0.000,B 0.000,C 90.000,E1 97.352} C_DIS
LIN {X 0.048,Y -482.174,Z 1304.540,A 0.000,B 0.000,C 90.000,E1 97.125} C_DIS
LIN {X -0.068,Y -480.734,Z 1304.538,A 0.000,B 0.000,C 90.000,E1 96.891} C_DIS
LIN {X 0.184,Y -467.716,Z 1304.528,A 0.000,B 0.000,C 90.000,E1 95.106} C_DIS
LIN {X -0.055,Y -453.978,Z 1304.517,A 0.000,B 0.000,C 90.000,E1 93.094} C_DIS
LIN {X -0.012,Y -438.996,Z 1304.504,A 0.000,B 0.000,C 90.000,E1 90.745} C_DIS
LIN {X 0.043,Y -421.206,Z 1304.486,A 0.000,B 0.000,C 90.000,E1 87.535} C_DIS
LIN {X 0.034,Y -409.653,Z 1304.474,A 0.000,B 0.000,C 90.000,E1 85.355} C_DIS
LIN {X 0.099,Y -400.846,Z 1304.465,A 0.000,B 0.000,C 90.000,E1 83.685} C_DIS
LIN {X 0.059,Y -390.480,Z 1304.454,A 0.000,B 0.000,C 90.000,E1 81.724} C_DIS
LIN {X -0.108,Y -381.287,Z 1304.445,A 0.000,B 0.000,C 90.000,E1 80.038} C_DIS
LIN {X 0.008,Y -371.709,Z 1304.435,A 0.000,B 0.000,C 90.000,E1 78.285} C_DIS
LIN {X 0.029,Y -362.010,Z 1304.425,A 0.000,B 0.000,C 90.000,E1 76.520} C_DIS
LIN {X -0.090,Y -350.464,Z 1304.414,A 0.000,B 0.000,C 90.000,E1 74.448} C_DIS
LIN {X 0.065,Y -340.516,Z 1304.403,A 0.000,B 0.000,C 90.000,E1 72.598} C_DIS
LIN {X 0.079,Y -327.302,Z 1304.390,A 0.000,B 0.000,C 90.000,E1 70.115} C_DIS
LIN {X 0.149,Y -311.666,Z 1304.372,A 0.000,B 0.000,C 90.000,E1 66.922} C_DIS
LIN {X -0.058,Y -298.659,Z 1304.356,A 0.000,B 0.000,C 90.000,E1 64.024} C_DIS
LIN {X -0.035,Y -290.954,Z 1304.345,A 0.000,B 0.000,C 90.000,E1 62.025} C_DIS
LIN {X -0.042,Y -283.020,Z 1304.331,A 0.000,B 0.000,C 90.000,E1 59.665} C_DIS
LIN {X 0.075,Y -272.963,Z 1304.312,A 0.000,B 0.000,C 90.000,E1 56.215} C_DIS
LIN {X -0.110,Y -263.799,Z 1304.293,A 0.000,B 0.000,C 90.000,E1 52.763} C_DIS
LIN {X -0.026,Y -256.849,Z 1304.277,A 0.000,B 0.000,C 90.000,E1 49.908} C_DIS
LIN {X 0.009,Y -250.100,Z 1304.261,A 0.000,B 0.000,C 90.000,E1 47.025} C_DIS
LIN {X 0.021,Y -243.570,Z 1304.245,A 0.000,B 0.000,C 90.000,E1 44.109} C_DIS
LIN {X 0.012,Y -235.841,Z 1304.224,A 0.000,B 0.000,C 90.000,E1 40.415} C_DIS
LIN {X 0.006,Y -229.053,Z 1304.204,A 0.000,B 0.000,C 90.000,E1 36.664} C_DIS
LIN {X -0.074,Y -223.175,Z 1304.183,A 0.000,B 0.000,C 90.000,E1 32.880} C_DIS
LIN {X 0.046,Y -218.269,Z 1304.161,A 0.000,B 0.000,C 90.000,E1 28.999} C_DIS
LIN {X -0.123,Y -213.984,Z 1304.140,A 0.000,B 0.000,C 90.000,E1 25.155} C_DIS
LIN {X -0.101,Y -210.214,Z 1304.118,A 0.000,B 0.000,C 90.000,E1 21.227} C_DIS
LIN {X 0.086,Y -206.783,Z 1304.096,A 0.000,B 0.000,C 90.000,E1 17.221} C_DIS
LIN {X 0.062,Y -203.800,Z 1304.074,A 0.000,B 0.000,C 90.000,E1 13.244} C_DIS
LIN {X -0.003,Y -200.502,Z 1304.042,A 0.000,B 0.000,C 90.000,E1 7.644} C_DIS
LIN {X 0.086,Y -198.229,Z 1304.002,A 0.000,B 0.000,C 90.000,E1 0.344} C_DIS
LIN {X 0.004,Y -199.544,Z 1303.943,A 0.000,B 0.000,C 90.000,E1 349.803} C_DIS
LIN {X -0.005,Y -202.721,Z 1303.912,A 0.000,B 0.000,C 90.000,E1 344.157} C_DIS
LIN {X 0.046,Y -206.778,Z 1303.885,A 0.000,B 0.000,C 90.000,E1 339.337} C_DIS
LIN {X 0.079,Y -211.036,Z 1303.863,A 0.000,B 0.000,C 90.000,E1 335.357} C_DIS
LIN {X 0.037,Y -216.100,Z 1303.841,A 0.000,B 0.000,C 90.000,E1 331.435} C_DIS
LIN {X -0.102,Y -222.064,Z 1303.820,A 0.000,B 0.000,C 90.000,E1 327.582} C_DIS
LIN {X 0.051,Y -228.986,Z 1303.798,A 0.000,B 0.000,C 90.000,E1 323.703} C_DIS
LIN {X 0.099,Y -236.753,Z 1303.777,A 0.000,B 0.000,C 90.000,E1 319.908} C_DIS
LIN {X 0.023,Y -243.816,Z 1303.761,A 0.000,B 0.000,C 90.000,E1 316.944} C_DIS
LIN {X 0.112,Y -252.823,Z 1303.742,A 0.000,B 0.000,C 90.000,E1 313.623} C_DIS
LIN {X -0.110,Y -260.661,Z 1303.729,A 0.000,B 0.000,C 90.000,E1 311.148} C_DIS
LIN {X 0.078,Y -269.776,Z 1303.715,A 0.000,B 0.000,C 90.000,E1 308.624} C_DIS
LIN {X 0.110,Y -276.992,Z 1303.705,A 0.000,B 0.000,C 90.000,E1 306.870} C_DIS
LIN {X -0.074,Y -284.897,Z 1303.695,A 0.000,B 0.000,C 90.000,E1 305.185} C_DIS
LIN {X -0.156,Y -295.544,Z 1303.684,A 0.000,B 0.000,C 90.000,E1 303.166} C_DIS
LIN {X 0.012,Y -303.186,Z 1303.677,A 0.000,B 0.000,C 90.000,E1 301.799} C_DIS
LIN {X -0.156,Y -318.291,Z 1303.664,A 0.000,B 0.000,C 90.000,E1 299.539} C_DIS
LIN {X 0.038,Y -332.828,Z 1303.653,A 0.000,B 0.000,C 90.000,E1 297.590} C_DIS
LIN {X -0.215,Y -353.547,Z 1303.640,A 0.000,B 0.000,C 90.000,E1 295.155} C_DIS
LIN {X -0.133,Y -366.560,Z 1303.631,A 0.000,B 0.000,C 90.000,E1 293.643} C_DIS
LIN {X -0.035,Y -379.269,Z 1303.623,A 0.000,B 0.000,C 90.000,E1 292.153} C_DIS
LIN {X -0.232,Y -391.441,Z 1303.615,A 0.000,B 0.000,C 90.000,E1 290.737} C_DIS
LIN {X -0.062,Y -413.719,Z 1303.601,A 0.000,B 0.000,C 90.000,E1 288.181} C_DIS
LIN {X -0.098,Y -423.449,Z 1303.595,A 0.000,B 0.000,C 90.000,E1 287.094} C_DIS
LIN {X -0.193,Y -432.743,Z 1303.589,A 0.000,B 0.000,C 90.000,E1 286.024} C_DIS
LIN {X -0.139,Y -437.006,Z 1303.586,A 0.000,B 0.000,C 90.000,E1 285.481} C_DIS
LIN {X -0.174,Y -440.885,Z 1303.583,A 0.000,B 0.000,C 90.000,E1 284.954} C_DIS
LIN {X 0.150,Y -446.007,Z 1303.578,A 0.000,B 0.000,C 90.000,E1 284.120} C_DIS
LIN {X -0.026,Y -450.425,Z 1303.574,A 0.000,B 0.000,C 90.000,E1 283.355} C_DIS
LIN {X 0.097,Y -455.624,Z 1303.568,A 0.000,B 0.000,C 90.000,E1 282.299} C_DIS
LIN {X 0.184,Y -457.872,Z 1303.566,A 0.000,B 0.000,C 90.000,E1 281.771} C_DIS
LIN {X -0.168,Y -459.860,Z 1303.563,A 0.000,B 0.000,C 90.000,E1 281.299} C_DIS
LIN {X -0.151,Y -461.557,Z 1303.560,A 0.000,B 0.000,C 90.000,E1 280.782} C_DIS
LIN {X -0.035,Y -462.874,Z 1303.557,A 0.000,B 0.000,C 90.000,E1 280.254} C_DIS
LIN {X 0.089,Y -463.876,Z 1303.554,A 0.000,B 0.000,C 90.000,E1 279.726} C_DIS
LIN {X 0.143,Y -464.398,Z 1303.551,A 0.000,B 0.000,C 90.000,E1 279.208} C_DIS
LIN {X -0.254,Y -464.541,Z 1303.548,A 0.000,B 0.000,C 90.000,E1 278.746} C_DIS
LIN {X -0.119,Y -464.207,Z 1303.546,A 0.000,B 0.000,C 90.000,E1 278.219} C_DIS
LIN {X -0.051,Y -463.429,Z 1303.543,A 0.000,B 0.000,C 90.000,E1 277.701} C_DIS
LIN {X 0.017,Y -462.124,Z 1303.540,A 0.000,B 0.000,C 90.000,E1 277.182} C_DIS
LIN {X 0.081,Y -460.335,Z 1303.537,A 0.000,B 0.000,C 90.000,E1 276.663} C_DIS
LIN {X 0.136,Y -458.048,Z 1303.534,A 0.000,B 0.000,C 90.000,E1 276.144} C_DIS
LIN {X 0.175,Y -455.359,Z 1303.531,A 0.000,B 0.000,C 90.000,E1 275.625} C_DIS
LIN {X 0.198,Y -452.091,Z 1303.529,A 0.000,B 0.000,C 90.000,E1 275.106} C_DIS
LIN {X -0.043,Y -450.273,Z 1303.527,A 0.000,B 0.000,C 90.000,E1 274.878} C_DIS
LIN {X -0.046,Y -445.915,Z 1303.524,A 0.000,B 0.000,C 90.000,E1 274.359} C_DIS
LIN {X 0.151,Y -443.418,Z 1303.523,A 0.000,B 0.000,C 90.000,E1 274.073} C_DIS
LIN {X 0.150,Y -437.509,Z 1303.520,A 0.000,B 0.000,C 90.000,E1 273.555} C_DIS
LIN {X 0.205,Y -431.453,Z 1303.517,A 0.000,B 0.000,C 90.000,E1 273.094} C_DIS
LIN {X 0.170,Y -424.767,Z 1303.515,A 0.000,B 0.000,C 90.000,E1 272.694} C_DIS
LIN {X 0.167,Y -417.959,Z 1303.513,A 0.000,B 0.000,C 90.000,E1 272.350} C_DIS
LIN {X 0.124,Y -410.832,Z 1303.512,A 0.000,B 0.000,C 90.000,E1 272.064} C_DIS
LIN {X 0.058,Y -403.790,Z 1303.510,A 0.000,B 0.000,C 90.000,E1 271.835} C_DIS
LIN {X 0.121,Y -392.993,Z 1303.509,A 0.000,B 0.000,C 90.000,E1 271.547} C_DIS
LIN {X -0.088,Y -385.409,Z 1303.508,A 0.000,B 0.000,C 90.000,E1 271.432} C_DIS
LIN {X -0.103,Y -377.185,Z 1303.507,A 0.000,B 0.000,C 90.000,E1 271.318} C_DIS
LIN {X 0.030,Y -365.994,Z 1303.507,A 0.000,B 0.000,C 90.000,E1 271.203} C_DIS
LIN {X -0.163,Y -357.764,Z 1303.507,A 0.000,B 0.000,C 90.000,E1 271.203} C_DIS
LIN {X 0.066,Y -181.420,Z 1303.506,A 0.000,B 0.000,C 90.000,E1 271.146} C_DIS
LIN {X -0.073,Y -181.578,Z 1303.501,A 0.000,B 0.000,C 90.000,E1 270.172} C_DIS
LIN {X -0.069,Y -180.844,Z 1303.472,A 0.000,B 0.000,C 90.000,E1 264.951} C_DIS
LIN {X 0.013,Y -178.953,Z 1303.444,A 0.000,B 0.000,C 90.000,E1 259.859} C_DIS
LIN {X -0.094,Y -177.353,Z 1303.430,A 0.000,B 0.000,C 90.000,E1 257.353} C_DIS
LIN {X 0.002,Y -175.522,Z 1303.411,A 0.000,B 0.000,C 90.000,E1 253.921} C_DIS
LIN {X 0.004,Y -172.258,Z 1303.387,A 0.000,B 0.000,C 90.000,E1 249.645} C_DIS
LIN {X 0.042,Y -171.737,Z 1303.382,A 0.000,B 0.000,C 90.000,E1 248.773} C_DIS
LIN {X 0.051,Y -167.334,Z 1303.353,A 0.000,B 0.000,C 90.000,E1 243.589} C_DIS
LIN {X -0.017,Y -166.720,Z 1303.349,A 0.000,B 0.000,C 90.000,E1 242.743} C_DIS
LIN {X -0.019,Y -162.700,Z 1303.324,A 0.000,B 0.000,C 90.000,E1 238.377} C_DIS
LIN {X -0.042,Y -161.390,Z 1303.315,A 0.000,B 0.000,C 90.000,E1 236.628} C_DIS
LIN {X 0.000,Y -157.383,Z 1303.290,A 0.000,B 0.000,C 90.000,E1 232.190} C_DIS
LIN {X -0.066,Y -155.379,Z 1303.275,A 0.000,B 0.000,C 90.000,E1 229.542} C_DIS
LIN {X 0.081,Y -151.716,Z 1303.250,A 0.000,B 0.000,C 90.000,E1 225.000} C_DIS
LIN {X -0.011,Y -149.908,Z 1303.235,A 0.000,B 0.000,C 90.000,E1 222.324} C_DIS
LIN {X -0.092,Y -146.765,Z 1303.210,A 0.000,B 0.000,C 90.000,E1 217.810} C_DIS
LIN {X 0.012,Y -145.333,Z 1303.195,A 0.000,B 0.000,C 90.000,E1 215.025} C_DIS
LIN {X -0.072,Y -142.413,Z 1303.164,A 0.000,B 0.000,C 90.000,E1 209.539} C_DIS
LIN {X -0.022,Y -141.398,Z 1303.149,A 0.000,B 0.000,C 90.000,E1 206.744} C_DIS
LIN {X -0.035,Y -139.354,Z 1303.112,A 0.000,B 0.000,C 90.000,E1 200.248} C_DIS
LIN {X -0.047,Y -138.794,Z 1303.097,A 0.000,B 0.000,C 90.000,E1 197.457} C_DIS
LIN {X 0.008,Y -138.347,Z 1303.055,A 0.000,B 0.000,C 90.000,E1 189.962} C_DIS
LIN {X 0.025,Y -139.375,Z 1303.009,A 0.000,B 0.000,C 90.000,E1 181.547} C_DIS
LIN {X -0.062,Y -141.267,Z 1302.972,A 0.000,B 0.000,C 90.000,E1 175.065} C_DIS
LIN {X 0.038,Y -142.633,Z 1302.957,A 0.000,B 0.000,C 90.000,E1 172.243} C_DIS
LIN {X -0.011,Y -144.959,Z 1302.931,A 0.000,B 0.000,C 90.000,E1 167.645} C_DIS
LIN {X -0.020,Y -147.588,Z 1302.911,A 0.000,B 0.000,C 90.000,E1 163.976} C_DIS
LIN {X 0.010,Y -150.204,Z 1302.891,A 0.000,B 0.000,C 90.000,E1 160.315} C_DIS
LIN {X 0.078,Y -153.587,Z 1302.870,A 0.000,B 0.000,C 90.000,E1 156.666} C_DIS
LIN {X -0.073,Y -157.003,Z 1302.851,A 0.000,B 0.000,C 90.000,E1 153.127} C_DIS
LIN {X -0.001,Y -161.121,Z 1302.831,A 0.000,B 0.000,C 90.000,E1 149.537} C_DIS
LIN {X -0.056,Y -163.222,Z 1302.821,A 0.000,B 0.000,C 90.000,E1 147.788} C_DIS
LIN {X -0.052,Y -167.652,Z 1302.801,A 0.000,B 0.000,C 90.000,E1 144.276} C_DIS
LIN {X -0.038,Y -171.476,Z 1302.787,A 0.000,B 0.000,C 90.000,E1 141.662} C_DIS
LIN {X -0.108,Y -176.405,Z 1302.768,A 0.000,B 0.000,C 90.000,E1 138.243} C_DIS
LIN {X 0.014,Y -180.699,Z 1302.754,A 0.000,B 0.000,C 90.000,E1 135.648} C_DIS
LIN {X -0.005,Y -186.103,Z 1302.735,A 0.000,B 0.000,C 90.000,E1 132.285} C_DIS
LIN {X -0.069,Y -190.740,Z 1302.721,A 0.000,B 0.000,C 90.000,E1 129.806} C_DIS
LIN {X -0.038,Y -196.494,Z 1302.703,A 0.000,B 0.000,C 90.000,E1 126.503} C_DIS
LIN {X 0.047,Y -199.456,Z 1302.694,A 0.000,B 0.000,C 90.000,E1 124.978} C_DIS
LIN {X 0.038,Y -308.898,Z 1302.694,A 0.000,B 0.000,C 90.000,E1 124.978} C_DIS
LIN {X -0.019,Y -313.384,Z 1302.694,A 0.000,B 0.000,C 90.000,E1 124.865} C_DIS
LIN {X -0.027,Y -316.167,Z 1302.693,A 0.000,B 0.000,C 90.000,E1 124.692} C_DIS
LIN {X -0.110,Y -319.910,Z 1302.691,A 0.000,B 0.000,C 90.000,E1 124.326} C_DIS
LIN {X 0.188,Y -323.369,Z 1302.688,A 0.000,B 0.000,C 90.000,E1 123.706} C_DIS
LIN {X 0.000,Y -324.728,Z 1302.686,A 0.000,B 0.000,C 90.000,E1 123.420} C_DIS
LIN {X 0.077,Y -336.351,Z 1302.668,A 0.000,B 0.000,C 90.000,E1 120.256} C_DIS
LIN {X -0.141,Y -348.211,Z 1302.653,A 0.000,B 0.000,C 90.000,E1 117.513} C_DIS
LIN {X -0.026,Y -361.519,Z 1302.638,A 0.000,B 0.000,C 90.000,E1 114.771} C_DIS
LIN {X 0.070,Y -374.662,Z 1302.624,A 0.000,B 0.000,C 90.000,E1 112.386} C_DIS
LIN {X 0.077,Y -389.134,Z 1302.612,A 0.000,B 0.000,C 90.000,E1 110.066} C_DIS
LIN {X -0.055,Y -405.037,Z 1302.599,A 0.000,B 0.000,C 90.000,E1 107.819} C_DIS
LIN {X -0.048,Y -422.484,Z 1302.587,A 0.000,B 0.000,C 90.000,E1 105.607} C_DIS
LIN {X -0.127,Y -441.570,Z 1302.575,A 0.000,B 0.000,C 90.000,E1 103.467} C_DIS
LIN {X 0.118,Y -461.644,Z 1302.564,A 0.000,B 0.000,C 90.000,E1 101.422} C_DIS
LIN {X 0.146,Y -477.054,Z 1302.556,A 0.000,B 0.000,C 90.000,E1 100.018} C_DIS
LIN {X 0.142,Y -479.220,Z 1302.554,A 0.000,B 0.000,C 90.000,E1 99.792} C_DIS
LIN {X 0.016,Y -481.016,Z 1302.553,A 0.000,B 0.000,C 90.000,E1 99.557} C_DIS
LIN {X -0.113,Y -482.364,Z 1302.552,A 0.000,B 0.000,C 90.000,E1 99.321} C_DIS
LIN {X 0.051,Y -484.046,Z 1302.549,A 0.000,B 0.000,C 90.000,E1 98.803} C_DIS
LIN {X -0.252,Y -484.650,Z 1302.546,A 0.000,B 0.000,C 90.000,E1 98.341} C_DIS
LIN {X 0.001,Y -484.274,Z 1302.543,A 0.000,B 0.000,C 90.000,E1 97.814} C_DIS
LIN {X 0.189,Y -482.863,Z 1302.541,A 0.000,B 0.000,C 90.000,E1 97.296} C_DIS
LIN {X 0.013,Y -481.697,Z 1302.539,A 0.000,B 0.000,C 90.000,E1 97.068} C_DIS
LIN {X -0.102,Y -480.140,Z 1302.538,A 0.000,B 0.000,C 90.000,E1 96.834} C_DIS
LIN {X -0.125,Y -468.851,Z 1302.530,A 0.000,B 0.000,C 90.000,E1 95.334} C_DIS
LIN {X 0.095,Y -455.051,Z 1302.518,A 0.000,B 0.000,C 90.000,E1 93.269} C_DIS
LIN {X -0.082,Y -438.384,Z 1302.504,A 0.000,B 0.000,C 90.000,E1 90.688} C_DIS
LIN {X -0.045,Y -420.631,Z 1302.486,A 0.000,B 0.000,C 90.000,E1 87.478} C_DIS
LIN {X -0.065,Y -409.074,Z 1302.474,A 0.000,B 0.000,C 90.000,E1 85.298} C_DIS
LIN {X 0.071,Y -398.773,Z 1302.463,A 0.000,B 0.000,C 90.000,E1 83.337} C_DIS
LIN {X -0.004,Y -389.915,Z 1302.454,A 0.000,B 0.000,C 90.000,E1 81.659} C_DIS
LIN {X 0.138,Y -380.688,Z 1302.444,A 0.000,B 0.000,C 90.000,E1 79.926} C_DIS
LIN {X -0.130,Y -371.121,Z 1302.434,A 0.000,B 0.000,C 90.000,E1 78.229} C_DIS
LIN {X -0.119,Y -361.427,Z 1302.425,A 0.000,B 0.000,C 90.000,E1 76.464} C_DIS
LIN {X 0.089,Y -349.866,Z 1302.413,A 0.000,B 0.000,C 90.000,E1 74.338} C_DIS
LIN {X -0.103,Y -339.909,Z 1302.403,A 0.000,B 0.000,C 90.000,E1 72.543} C_DIS
LIN {X -0.101,Y -326.736,Z 1302.389,A 0.000,B 0.000,C 90.000,E1 70.061} C_DIS
LIN {X -0.046,Y -311.160,Z 1302.371,A 0.000,B 0.000,C 90.000,E1 66.869} C_DIS
LIN {X 0.135,Y -298.208,Z 1302.355,A 0.000,B 0.000,C 90.000,E1 63.896} C_DIS
LIN {X 0.145,Y -290.573,Z 1302.344,A 0.000,B 0.000,C 90.000,E1 61.897} C_DIS
LIN {X 0.124,Y -282.682,Z 1302.331,A 0.000,B 0.000,C 90.000,E1 59.537} C_DIS
LIN {X -0.005,Y -272.654,Z 1302.312,A 0.000,B 0.000,C 90.000,E1 56.135} C_DIS
LIN {X 0.017,Y -263.498,Z 1302.292,A 0.000,B 0.000,C 90.000,E1 52.637} C_DIS
LIN {X -0.112,Y -256.534,Z 1302.277,A 0.000,B 0.000,C 90.000,E1 49.828} C_DIS
LIN {X 0.089,Y -249.791,Z 1302.261,A 0.000,B 0.000,C 90.000,E1 46.905} C_DIS
LIN {X -0.075,Y -243.254,Z 1302.245,A 0.000,B 0.000,C 90.000,E1 44.028} C_DIS
LIN {X 0.061,Y -235.542,Z 1302.224,A 0.000,B 0.000,C 90.000,E1 40.297} C_DIS
LIN {X -0.106,Y -228.778,Z 1302.203,A 0.000,B 0.000,C 90.000,E1 36.583} C_DIS
LIN {X -0.007,Y -222.905,Z 1302.182,A 0.000,B 0.000,C 90.000,E1 32.752} C_DIS
LIN {X -0.001,Y -217.999,Z 1302.161,A 0.000,B 0.000,C 90.000,E1 28.899} C_DIS
LIN {X 0.068,Y -212.871,Z 1302.135,A 0.000,B 0.000,C 90.000,E1 24.207} C_DIS
LIN {X -0.031,Y -209.175,Z 1302.113,A 0.000,B 0.000,C 90.000,E1 20.301} C_DIS
LIN {X 0.051,Y -205.778,Z 1302.091,A 0.000,B 0.000,C 90.000,E1 16.315} C_DIS
LIN {X -0.062,Y -202.895,Z 1302.068,A 0.000,B 0.000,C 90.000,E1 12.355} C_DIS
LIN {X -0.038,Y -199.812,Z 1302.037,A 0.000,B 0.000,C 90.000,E1 6.720} C_DIS
LIN {X 0.000,Y -197.957,Z 1302.000,A 0.000,B 0.000,C 90.000,E1 360.000} C_DIS
LIN {X -0.010,Y -199.423,Z 1301.943,A 0.000,B 0.000,C 90.000,E1 349.803} C_DIS
LIN {X -0.023,Y -202.669,Z 1301.912,A 0.000,B 0.000,C 90.000,E1 344.157} C_DIS
LIN {X 0.026,Y -206.770,Z 1301.885,A 0.000,B 0.000,C 90.000,E1 339.337} C_DIS
LIN {X 0.058,Y -211.082,Z 1301.863,A 0.000,B 0.000,C 90.000,E1 335.357} C_DIS
LIN {X 0.017,Y -216.166,Z 1301.841,A 0.000,B 0.000,C 90.000,E1 331.435} C_DIS
LIN {X 0.068,Y -222.140,Z 1301.820,A 0.000,B 0.000,C 90.000,E1 327.533} C_DIS
LIN {X 0.035,Y -229.049,Z 1301.798,A 0.000,B 0.000,C 90.000,E1 323.703} C_DIS
LIN {X 0.085,Y -236.810,Z 1301.777,A 0.000,B 0.000,C 90.000,E1 319.908} C_DIS
LIN {X 0.009,Y -243.878,Z 1301.761,A 0.000,B 0.000,C 90.000,E1 316.944} C_DIS
LIN {X 0.099,Y -252.863,Z 1301.742,A 0.000,B 0.000,C 90.000,E1 313.623} C_DIS
LIN {X 0.037,Y -259.495,Z 1301.730,A 0.000,B 0.000,C 90.000,E1 311.472} C_DIS
LIN {X -0.130,Y -265.750,Z 1301.721,A 0.000,B 0.000,C 90.000,E1 309.725} C_DIS
LIN {X 0.007,Y -275.490,Z 1301.707,A 0.000,B 0.000,C 90.000,E1 307.237} C_DIS
LIN {X -0.087,Y -284.912,Z 1301.695,A 0.000,B 0.000,C 90.000,E1 305.185} C_DIS
LIN {X -0.168,Y -295.574,Z 1301.684,A 0.000,B 0.000,C 90.000,E1 303.166} C_DIS
LIN {X -0.001,Y -303.208,Z 1301.677,A 0.000,B 0.000,C 90.000,E1 301.799} C_DIS
LIN {X -0.168,Y -318.293,Z 1301.664,A 0.000,B 0.000,C 90.000,E1 299.539} C_DIS
LIN {X 0.025,Y -332.824,Z 1301.653,A 0.000,B 0.000,C 90.000,E1 297.590} C_DIS
LIN {X 0.093,Y -353.510,Z 1301.640,A 0.000,B 0.000,C 90.000,E1 295.103} C_DIS
LIN {X 0.089,Y -366.197,Z 1301.631,A 0.000,B 0.000,C 90.000,E1 293.643} C_DIS
LIN {X -0.162,Y -378.926,Z 1301.623,A 0.000,B 0.000,C 90.000,E1 292.206} C_DIS
LIN {X -0.005,Y -391.139,Z 1301.615,A 0.000,B 0.000,C 90.000,E1 290.737} C_DIS
LIN {X 0.200,Y -413.368,Z 1301.601,A 0.000,B 0.000,C 90.000,E1 288.181} C_DIS
LIN {X 0.119,Y -423.173,Z 1301.595,A 0.000,B 0.000,C 90.000,E1 287.094} C_DIS
LIN {X 0.027,Y -432.520,Z 1301.589,A 0.000,B 0.000,C 90.000,E1 286.024} C_DIS
LIN {X -0.148,Y -438.808,Z 1301.585,A 0.000,B 0.000,C 90.000,E1 285.245} C_DIS
LIN {X 0.039,Y -444.251,Z 1301.580,A 0.000,B 0.000,C 90.000,E1 284.426} C_DIS
LIN {X -0.038,Y -448.935,Z 1301.576,A 0.000,B 0.000,C 90.000,E1 283.647} C_DIS
LIN {X 0.065,Y -454.342,Z 1301.570,A 0.000,B 0.000,C 90.000,E1 282.591} C_DIS
LIN {X -0.038,Y -457.840,Z 1301.566,A 0.000,B 0.000,C 90.000,E1 281.827} C_DIS
LIN {X 0.059,Y -459.857,Z 1301.563,A 0.000,B 0.000,C 90.000,E1 281.299} C_DIS
LIN {X 0.076,Y -461.565,Z 1301.560,A 0.000,B 0.000,C 90.000,E1 280.782} C_DIS
LIN {X 0.193,Y -462.956,Z 1301.557,A 0.000,B 0.000,C 90.000,E1 280.254} C_DIS
LIN {X -0.140,Y -463.940,Z 1301.554,A 0.000,B 0.000,C 90.000,E1 279.782} C_DIS
LIN {X -0.086,Y -464.535,Z 1301.551,A 0.000,B 0.000,C 90.000,E1 279.265} C_DIS
LIN {X -0.023,Y -464.721,Z 1301.549,A 0.000,B 0.000,C 90.000,E1 278.746} C_DIS
LIN {X 0.112,Y -464.442,Z 1301.546,A 0.000,B 0.000,C 90.000,E1 278.219} C_DIS
LIN {X 0.181,Y -463.657,Z 1301.543,A 0.000,B 0.000,C 90.000,E1 277.701} C_DIS
LIN {X -0.209,Y -462.435,Z 1301.540,A 0.000,B 0.000,C 90.000,E1 277.239} C_DIS
LIN {X 0.139,Y -459.675,Z 1301.536,A 0.000,B 0.000,C 90.000,E1 276.429} C_DIS
LIN {X 0.186,Y -457.274,Z 1301.533,A 0.000,B 0.000,C 90.000,E1 275.910} C_DIS
LIN {X 0.217,Y -454.374,Z 1301.530,A 0.000,B 0.000,C 90.000,E1 275.391} C_DIS
LIN {X 0.193,Y -450.940,Z 1301.527,A 0.000,B 0.000,C 90.000,E1 274.878} C_DIS
LIN {X 0.190,Y -446.720,Z 1301.524,A 0.000,B 0.000,C 90.000,E1 274.359} C_DIS
LIN {X -0.054,Y -444.309,Z 1301.523,A 0.000,B 0.000,C 90.000,E1 274.131} C_DIS
LIN {X -0.090,Y -438.491,Z 1301.520,A 0.000,B 0.000,C 90.000,E1 273.612} C_DIS
LIN {X -0.084,Y -432.484,Z 1301.517,A 0.000,B 0.000,C 90.000,E1 273.154} C_DIS
LIN {X -0.108,Y -425.990,Z 1301.515,A 0.000,B 0.000,C 90.000,E1 272.751} C_DIS
LIN {X -0.118,Y -419.306,Z 1301.513,A 0.000,B 0.000,C 90.000,E1 272.407} C_DIS
LIN {X -0.180,Y -412.319,Z 1301.512,A 0.000,B 0.000,C 90.000,E1 272.121} C_DIS
LIN {X 0.108,Y -405.190,Z 1301.510,A 0.000,B 0.000,C 90.000,E1 271.835} C_DIS
LIN {X -0.134,Y -397.813,Z 1301.509,A 0.000,B 0.000,C 90.000,E1 271.661} C_DIS
LIN {X -0.118,Y -390.173,Z 1301.508,A 0.000,B 0.000,C 90.000,E1 271.489} C_DIS
LIN {X 0.153,Y -378.066,Z 1301.507,A 0.000,B 0.000,C 90.000,E1 271.260} C_DIS
LIN {X -0.096,Y -367.368,Z 1301.507,A 0.000,B 0.000,C 90.000,E1 271.203} C_DIS
LIN {X -0.004,Y -355.397,Z 1301.506,A 0.000,B 0.000,C 90.000,E1 271.146} C_DIS
LIN {X -0.020,Y -181.425,Z 1301.506,A 0.000,B 0.000,C 90.000,E1 271.146} C_DIS
LIN {X 0.089,Y -181.581,Z 1301.501,A 0.000,B 0.000,C 90.000,E1 270.229} C_DIS
LIN {X 0.078,Y -180.896,Z 1301.473,A 0.000,B 0.000,C 90.000,E1 265.179} C_DIS
LIN {X 0.084,Y -179.841,Z 1301.459,A 0.000,B 0.000,C 90.000,E1 262.648} C_DIS
LIN {X -0.038,Y -179.026,Z 1301.445,A 0.000,B 0.000,C 90.000,E1 260.151} C_DIS
LIN {X 0.024,Y -178.671,Z 1301.441,A 0.000,B 0.000,C 90.000,E1 259.285} C_DIS
LIN {X -0.040,Y -175.721,Z 1301.412,A 0.000,B 0.000,C 90.000,E1 254.212} C_DIS
LIN {X -0.023,Y -172.437,Z 1301.388,A 0.000,B 0.000,C 90.000,E1 249.934} C_DIS
LIN {X -0.067,Y -171.267,Z 1301.379,A 0.000,B 0.000,C 90.000,E1 248.230} C_DIS
LIN {X -0.021,Y -167.537,Z 1301.355,A 0.000,B 0.000,C 90.000,E1 243.896} C_DIS
LIN {X -0.007,Y -166.152,Z 1301.345,A 0.000,B 0.000,C 90.000,E1 242.153} C_DIS
LIN {X -0.017,Y -162.928,Z 1301.326,A 0.000,B 0.000,C 90.000,E1 238.663} C_DIS
LIN {X -0.039,Y -161.601,Z 1301.316,A 0.000,B 0.000,C 90.000,E1 236.914} C_DIS
LIN {X 0.086,Y -158.345,Z 1301.297,A 0.000,B 0.000,C 90.000,E1 233.336} C_DIS
LIN {X -0.052,Y -155.647,Z 1301.277,A 0.000,B 0.000,C 90.000,E1 229.828} C_DIS
LIN {X 0.001,Y -151.919,Z 1301.252,A 0.000,B 0.000,C 90.000,E1 225.324} C_DIS
LIN {X 0.016,Y -150.153,Z 1301.237,A 0.000,B 0.000,C 90.000,E1 222.609} C_DIS
LIN {X -0.063,Y -146.936,Z 1301.212,A 0.000,B 0.000,C 90.000,E1 218.096} C_DIS
LIN {X 0.043,Y -145.523,Z 1301.196,A 0.000,B 0.000,C 90.000,E1 215.311} C_DIS
LIN {X 0.038,Y -142.923,Z 1301.171,A 0.000,B 0.000,C 90.000,E1 210.718} C_DIS
LIN {X -0.036,Y -141.545,Z 1301.150,A 0.000,B 0.000,C 90.000,E1 207.052} C_DIS
LIN {X -0.047,Y -139.403,Z 1301.114,A 0.000,B 0.000,C 90.000,E1 200.556} C_DIS
LIN {X 0.007,Y -139.121,Z 1301.104,A 0.000,B 0.000,C 90.000,E1 198.671} C_DIS
LIN {X 0.038,Y -138.351,Z 1301.057,A 0.000,B 0.000,C 90.000,E1 190.254} C_DIS
LIN {X 0.029,Y -139.502,Z 1301.005,A 0.000,B 0.000,C 90.000,E1 180.917} C_DIS
LIN {X -0.031,Y -141.133,Z 1300.974,A 0.000,B 0.000,C 90.000,E1 175.355} C_DIS
LIN {X -0.078,Y -142.514,Z 1300.959,A 0.000,B 0.000,C 90.000,E1 172.591} C_DIS
LIN {X 0.009,Y -144.774,Z 1300.933,A 0.000,B 0.000,C 90.000,E1 167.937} C_DIS
LIN {X -0.042,Y -147.388,Z 1300.913,A 0.000,B 0.000,C 90.000,E1 164.283} C_DIS
LIN {X 0.021,Y -150.718,Z 1300.887,A 0.000,B 0.000,C 90.000,E1 159.699} C_DIS
LIN {X -0.039,Y -154.199,Z 1300.867,A 0.000,B 0.000,C 90.000,E1 156.102} C_DIS
LIN {X 0.030,Y -157.638,Z 1300.847,A 0.000,B 0.000,C 90.000,E1 152.487} C_DIS
LIN {X -0.022,Y -161.896,Z 1300.827,A 0.000,B 0.000,C 90.000,E1 148.948} C_DIS
LIN {X 0.086,Y -166.087,Z 1300.808,A 0.000,B 0.000,C 90.000,E1 145.388} C_DIS
LIN {X 0.085,Y -171.095,Z 1300.788,A 0.000,B 0.000,C 90.000,E1 141.904} C_DIS
LIN {X 0.005,Y -175.970,Z 1300.769,A 0.000,B 0.000,C 90.000,E1 138.485} C_DIS
LIN {X 0.119,Y -180.215,Z 1300.755,A 0.000,B 0.000,C 90.000,E1 135.891} C_DIS
LIN {X 0.093,Y -185.629,Z 1300.736,A 0.000,B 0.000,C 90.000,E1 132.528} C_DIS
LIN {X -0.121,Y -190.225,Z 1300.723,A 0.000,B 0.000,C 90.000,E1 130.092} C_DIS
LIN {X 0.038,Y -197.553,Z 1300.700,A 0.000,B 0.000,C 90.000,E1 125.931} C_DIS
LIN {X -0.025,Y -199.498,Z 1300.694,A 0.000,B 0.000,C 90.000,E1 124.978} C_DIS
LIN {X 0.090,Y -309.601,Z 1300.694,A 0.000,B 0.000,C 90.000,E1 124.945} C_DIS
LIN {X -0.059,Y -311.029,Z 1300.694,A 0.000,B 0.000,C 90.000,E1 124.945} C_DIS
LIN {X 0.071,Y -316.763,Z 1300.692,A 0.000,B 0.000,C 90.000,E1 124.612} C_DIS
LIN {X -0.058,Y -319.744,Z 1300.691,A 0.000,B 0.000,C 90.000,E1 124.326} C_DIS
LIN {X -0.068,Y -321.752,Z 1300.689,A 0.000,B 0.000,C 90.000,E1 124.040} C_DIS
LIN {X 0.190,Y -323.323,Z 1300.688,A 0.000,B 0.000,C 90.000,E1 123.706} C_DIS
LIN {X 0.007,Y -324.695,Z 1300.686,A 0.000,B 0.000,C 90.000,E1 123.420} C_DIS
LIN {X 0.090,Y -336.321,Z 1300.668,A 0.000,B 0.000,C 90.000,E1 120.256} C_DIS
LIN {X -0.128,Y -348.179,Z 1300.653,A 0.000,B 0.000,C 90.000,E1 117.513} C_DIS
LIN {X -0.014,Y -361.485,Z 1300.638,A 0.000,B 0.000,C 90.000,E1 114.771} C_DIS
LIN {X 0.082,Y -374.627,Z 1300.624,A 0.000,B 0.000,C 90.000,E1 112.386} C_DIS
LIN {X 0.088,Y -389.098,Z 1300.612,A 0.000,B 0.000,C 90.000,E1 110.066} C_DIS
LIN {X -0.044,Y -405.000,Z 1300.599,A 0.000,B 0.000,C 90.000,E1 107.819} C_DIS
LIN {X -0.038,Y -422.445,Z 1300.587,A 0.000,B 0.000,C 90.000,E1 105.607} C_DIS
LIN {X -0.117,Y -441.531,Z 1300.575,A 0.000,B 0.000,C 90.000,E1 103.467} C_DIS
LIN {X 0.126,Y -461.603,Z 1300.564,A 0.000,B 0.000,C 90.000,E1 101.422} C_DIS
LIN {X 0.152,Y -477.010,Z 1300.556,A 0.000,B 0.000,C 90.000,E1 100.018} C_DIS
LIN {X 0.149,Y -479.154,Z 1300.554,A 0.000,B 0.000,C 90.000,E1 99.792} C_DIS
LIN {X 0.022,Y -480.934,Z 1300.553,A 0.000,B 0.000,C 90.000,E1 99.557} C_DIS
LIN {X -0.106,Y -482.270,Z 1300.552,A 0.000,B 0.000,C 90.000,E1 99.321} C_DIS
LIN {X 0.058,Y -483.934,Z 1300.549,A 0.000,B 0.000,C 90.000,E1 98.803} C_DIS
LIN {X -0.246,Y -484.521,Z 1300.546,A 0.000,B 0.000,C 90.000,E1 98.341} C_DIS
LIN {X 0.006,Y -484.130,Z 1300.543,A 0.000,B 0.000,C 90.000,E1 97.814} C_DIS
LIN {X 0.194,Y -482.702,Z 1300.541,A 0.000,B 0.000,C 90.000,E1 97.296} C_DIS
LIN {X 0.017,Y -481.527,Z 1300.539,A 0.000,B 0.000,C 90.000,E1 97.068} C_DIS
LIN {X -0.098,Y -479.956,Z 1300.538,A 0.000,B 0.000,C 90.000,E1 96.834} C_DIS
LIN {X -0.124,Y -468.669,Z 1300.530,A 0.000,B 0.000,C 90.000,E1 95.334} C_DIS
LIN {X 0.091,Y -454.838,Z 1300.518,A 0.000,B 0.000,C 90.000,E1 93.269} C_DIS
LIN {X -0.092,Y -438.163,Z 1300.504,A 0.000,B 0.000,C 90.000,E1 90.688} C_DIS
LIN {X -0.062,Y -420.401,Z 1300.486,A 0.000,B 0.000,C 90.000,E1 87.478} C_DIS
LIN {X -0.088,Y -408.849,Z 1300.474,A 0.000,B 0.000,C 90.000,E1 85.298} C_DIS
LIN {X -0.035,Y -400.034,Z 1300.465,A 0.000,B 0.000,C 90.000,E1 83.628} C_DIS
LIN {X -0.033,Y -389.683,Z 1300.454,A 0.000,B 0.000,C 90.000,E1 81.659} C_DIS
LIN {X 0.105,Y -380.474,Z 1300.444,A 0.000,B 0.000,C 90.000,E1 79.926} C_DIS
LIN {X -0.165,Y -370.938,Z 1300.434,A 0.000,B 0.000,C 90.000,E1 78.229} C_DIS
LIN {X -0.156,Y -361.238,Z 1300.425,A 0.000,B 0.000,C 90.000,E1 76.464} C_DIS
LIN {X 0.048,Y -349.668,Z 1300.413,A 0.000,B 0.000,C 90.000,E1 74.338} C_DIS
LIN {X -0.146,Y -339.712,Z 1300.403,A 0.000,B 0.000,C 90.000,E1 72.543} C_DIS
LIN {X -0.148,Y -326.565,Z 1300.389,A 0.000,B 0.000,C 90.000,E1 70.061} C_DIS
LIN {X -0.053,Y -309.525,Z 1300.370,A 0.000,B 0.000,C 90.000,E1 66.538} C_DIS
LIN {X 0.085,Y -298.103,Z 1300.355,A 0.000,B 0.000,C 90.000,E1 63.896} C_DIS
LIN {X 0.094,Y -290.490,Z 1300.344,A 0.000,B 0.000,C 90.000,E1 61.897} C_DIS
LIN {X 0.073,Y -282.604,Z 1300.331,A 0.000,B 0.000,C 90.000,E1 59.537} C_DIS
LIN {X -0.057,Y -272.580,Z 1300.312,A 0.000,B 0.000,C 90.000,E1 56.135} C_DIS
LIN {X -0.035,Y -263.406,Z 1300.292,A 0.000,B 0.000,C 90.000,E1 52.637} C_DIS
LIN {X 0.031,Y -256.432,Z 1300.277,A 0.000,B 0.000,C 90.000,E1 49.784} C_DIS
LIN {X 0.035,Y -249.671,Z 1300.261,A 0.000,B 0.000,C 90.000,E1 46.905} C_DIS
LIN {X -0.131,Y -243.129,Z 1300.244,A 0.000,B 0.000,C 90.000,E1 44.028} C_DIS
LIN {X 0.003,Y -235.417,Z 1300.224,A 0.000,B 0.000,C 90.000,E1 40.297} C_DIS
LIN {X 0.017,Y -228.642,Z 1300.203,A 0.000,B 0.000,C 90.000,E1 36.537} C_DIS
LIN {X -0.071,Y -222.754,Z 1300.182,A 0.000,B 0.000,C 90.000,E1 32.752} C_DIS
LIN {X 0.039,Y -217.830,Z 1300.160,A 0.000,B 0.000,C 90.000,E1 28.871} C_DIS
LIN {X -0.004,Y -212.646,Z 1300.135,A 0.000,B 0.000,C 90.000,E1 24.207} C_DIS
LIN {X 0.087,Y -208.899,Z 1300.113,A 0.000,B 0.000,C 90.000,E1 20.248} C_DIS
LIN {X -0.035,Y -205.481,Z 1300.091,A 0.000,B 0.000,C 90.000,E1 16.315} C_DIS
LIN {X 0.043,Y -202.596,Z 1300.068,A 0.000,B 0.000,C 90.000,E1 12.299} C_DIS
LIN {X 0.055,Y -199.528,Z 1300.037,A 0.000,B 0.000,C 90.000,E1 6.663} C_DIS
LIN {X 0.000,Y -197.732,Z 1300.000,A 0.000,B 0.000,C 90.000,E1 360.000} C_DIS
LIN {X -0.024,Y -199.292,Z 1299.943,A 0.000,B 0.000,C 90.000,E1 349.803} C_DIS
LIN {X -0.043,Y -202.623,Z 1299.912,A 0.000,B 0.000,C 90.000,E1 344.157} C_DIS
LIN {X 0.005,Y -206.762,Z 1299.885,A 0.000,B 0.000,C 90.000,E1 339.337} C_DIS
LIN {X 0.037,Y -211.124,Z 1299.863,A 0.000,B 0.000,C 90.000,E1 335.357} C_DIS
LIN {X -0.004,Y -216.232,Z 1299.841,A 0.000,B 0.000,C 90.000,E1 331.435} C_DIS
LIN {X 0.049,Y -222.204,Z 1299.820,A 0.000,B 0.000,C 90.000,E1 327.533} C_DIS
LIN {X 0.018,Y -229.093,Z 1299.798,A 0.000,B 0.000,C 90.000,E1 323.703} C_DIS
LIN {X 0.068,Y -236.869,Z 1299.777,A 0.000,B 0.000,C 90.000,E1 319.908} C_DIS
LIN {X -0.007,Y -243.922,Z 1299.761,A 0.000,B 0.000,C 90.000,E1 316.944} C_DIS
LIN {X 0.084,Y -252.896,Z 1299.742,A 0.000,B 0.000,C 90.000,E1 313.623} C_DIS
LIN {X 0.022,Y -259.516,Z 1299.730,A 0.000,B 0.000,C 90.000,E1 311.472} C_DIS
LIN {X -0.145,Y -265.759,Z 1299.720,A 0.000,B 0.000,C 90.000,E1 309.725} C_DIS
LIN {X -0.008,Y -275.491,Z 1299.707,A 0.000,B 0.000,C 90.000,E1 307.237} C_DIS
LIN {X 0.061,Y -284.919,Z 1299.695,A 0.000,B 0.000,C 90.000,E1 305.152} C_DIS
LIN {X -0.185,Y -295.561,Z 1299.684,A 0.000,B 0.000,C 90.000,E1 303.166} C_DIS
LIN {X -0.018,Y -303.213,Z 1299.677,A 0.000,B 0.000,C 90.000,E1 301.799} C_DIS
LIN {X -0.186,Y -318.305,Z 1299.664,A 0.000,B 0.000,C 90.000,E1 299.539} C_DIS
LIN {X 0.061,Y -330.293,Z 1299.655,A 0.000,B 0.000,C 90.000,E1 297.897} C_DIS
LIN {X 0.067,Y -350.850,Z 1299.641,A 0.000,B 0.000,C 90.000,E1 295.412} C_DIS
LIN {X 0.024,Y -363.584,Z 1299.633,A 0.000,B 0.000,C 90.000,E1 293.951} C_DIS
LIN {X 0.086,Y -376.336,Z 1299.625,A 0.000,B 0.000,C 90.000,E1 292.461} C_DIS
LIN {X 0.208,Y -386.263,Z 1299.618,A 0.000,B 0.000,C 90.000,E1 291.280} C_DIS
LIN {X 0.053,Y -405.769,Z 1299.606,A 0.000,B 0.000,C 90.000,E1 289.033} C_DIS
LIN {X -0.151,Y -418.183,Z 1299.598,A 0.000,B 0.000,C 90.000,E1 287.692} C_DIS
LIN {X 0.081,Y -430.017,Z 1299.591,A 0.000,B 0.000,C 90.000,E1 286.315} C_DIS
LIN {X -0.122,Y -436.601,Z 1299.586,A 0.000,B 0.000,C 90.000,E1 285.536} C_DIS
LIN {X 0.046,Y -442.409,Z 1299.582,A 0.000,B 0.000,C 90.000,E1 284.717} C_DIS
LIN {X -0.054,Y -447.377,Z 1299.577,A 0.000,B 0.000,C 90.000,E1 283.939} C_DIS
LIN {X 0.224,Y -451.712,Z 1299.573,A 0.000,B 0.000,C 90.000,E1 283.119} C_DIS
LIN {X 0.099,Y -455.551,Z 1299.569,A 0.000,B 0.000,C 90.000,E1 282.355} C_DIS
LIN {X 0.008,Y -458.879,Z 1299.564,A 0.000,B 0.000,C 90.000,E1 281.591} C_DIS
LIN {X -0.146,Y -461.577,Z 1299.560,A 0.000,B 0.000,C 90.000,E1 280.838} C_DIS
LIN {X -0.030,Y -463.000,Z 1299.557,A 0.000,B 0.000,C 90.000,E1 280.310} C_DIS
LIN {X 0.014,Y -464.046,Z 1299.554,A 0.000,B 0.000,C 90.000,E1 279.792} C_DIS
LIN {X 0.147,Y -464.700,Z 1299.552,A 0.000,B 0.000,C 90.000,E1 279.265} C_DIS
LIN {X -0.250,Y -464.890,Z 1299.549,A 0.000,B 0.000,C 90.000,E1 278.803} C_DIS
LIN {X -0.113,Y -464.659,Z 1299.546,A 0.000,B 0.000,C 90.000,E1 278.276} C_DIS
LIN {X -0.045,Y -463.947,Z 1299.543,A 0.000,B 0.000,C 90.000,E1 277.757} C_DIS
LIN {X 0.025,Y -462.749,Z 1299.540,A 0.000,B 0.000,C 90.000,E1 277.239} C_DIS
LIN {X 0.092,Y -461.067,Z 1299.537,A 0.000,B 0.000,C 90.000,E1 276.720} C_DIS
LIN {X -0.029,Y -457.731,Z 1299.533,A 0.000,B 0.000,C 90.000,E1 275.967} C_DIS
LIN {X -0.034,Y -454.931,Z 1299.530,A 0.000,B 0.000,C 90.000,E1 275.454} C_DIS
LIN {X -0.011,Y -451.604,Z 1299.527,A 0.000,B 0.000,C 90.000,E1 274.935} C_DIS
LIN {X -0.009,Y -447.528,Z 1299.525,A 0.000,B 0.000,C 90.000,E1 274.416} C_DIS
LIN {X 0.193,Y -445.200,Z 1299.523,A 0.000,B 0.000,C 90.000,E1 274.131} C_DIS
LIN {X 0.159,Y -439.560,Z 1299.520,A 0.000,B 0.000,C 90.000,E1 273.612} C_DIS
LIN {X 0.100,Y -433.573,Z 1299.518,A 0.000,B 0.000,C 90.000,E1 273.154} C_DIS
LIN {X -0.124,Y -430.591,Z 1299.516,A 0.000,B 0.000,C 90.000,E1 272.980} C_DIS
LIN {X 0.041,Y -424.033,Z 1299.514,A 0.000,B 0.000,C 90.000,E1 272.579} C_DIS
LIN {X 0.163,Y -417.306,Z 1299.513,A 0.000,B 0.000,C 90.000,E1 272.236} C_DIS
LIN {X -0.195,Y -410.215,Z 1299.511,A 0.000,B 0.000,C 90.000,E1 272.007} C_DIS
LIN {X -0.190,Y -403.056,Z 1299.510,A 0.000,B 0.000,C 90.000,E1 271.776} C_DIS
LIN {X -0.123,Y -391.851,Z 1299.508,A 0.000,B 0.000,C 90.000,E1 271.489} C_DIS
LIN {X 0.072,Y -383.553,Z 1299.507,A 0.000,B 0.000,C 90.000,E1 271.318} C_DIS
LIN {X 0.112,Y -375.078,Z 1299.507,A 0.000,B 0.000,C 90.000,E1 271.203} C_DIS
LIN {X -0.096,Y -360.946,Z 1299.506,A 0.000,B 0.000,C 90.000,E1 271.146} C_DIS
LIN {X -0.142,Y -358.061,Z 1299.506,A 0.000,B 0.000,C 90.000,E1 271.146} C_DIS
LIN {X 0.085,Y -181.430,Z 1299.506,A 0.000,B 0.000,C 90.000,E1 271.088} C_DIS
LIN {X -0.002,Y -181.580,Z 1299.501,A 0.000,B 0.000,C 90.000,E1 270.229} C_DIS
LIN {X -0.013,Y -180.893,Z 1299.473,A 0.000,B 0.000,C 90.000,E1 265.179} C_DIS
LIN {X 0.064,Y -179.516,Z 1299.454,A 0.000,B 0.000,C 90.000,E1 261.781} C_DIS
LIN {X 0.049,Y -179.019,Z 1299.445,A 0.000,B 0.000,C 90.000,E1 260.095} C_DIS
LIN {X -0.032,Y -178.652,Z 1299.440,A 0.000,B 0.000,C 90.000,E1 259.275} C_DIS
LIN {X 0.041,Y -175.702,Z 1299.412,A 0.000,B 0.000,C 90.000,E1 254.157} C_DIS
LIN {X 0.051,Y -172.418,Z 1299.388,A 0.000,B 0.000,C 90.000,E1 249.880} C_DIS
LIN {X 0.067,Y -171.238,Z 1299.379,A 0.000,B 0.000,C 90.000,E1 248.156} C_DIS
LIN {X 0.043,Y -167.516,Z 1299.355,A 0.000,B 0.000,C 90.000,E1 243.845} C_DIS
LIN {X -0.024,Y -166.911,Z 1299.350,A 0.000,B 0.000,C 90.000,E1 242.999} C_DIS
LIN {X 0.027,Y -162.219,Z 1299.321,A 0.000,B 0.000,C 90.000,E1 237.740} C_DIS
LIN {X -0.053,Y -160.800,Z 1299.311,A 0.000,B 0.000,C 90.000,E1 236.008} C_DIS
LIN {X -0.074,Y -157.588,Z 1299.291,A 0.000,B 0.000,C 90.000,E1 232.477} C_DIS
LIN {X -0.016,Y -155.621,Z 1299.276,A 0.000,B 0.000,C 90.000,E1 229.784} C_DIS
LIN {X -0.081,Y -151.898,Z 1299.252,A 0.000,B 0.000,C 90.000,E1 225.324} C_DIS
LIN {X -0.065,Y -150.127,Z 1299.237,A 0.000,B 0.000,C 90.000,E1 222.609} C_DIS
LIN {X 0.063,Y -146.918,Z 1299.211,A 0.000,B 0.000,C 90.000,E1 218.016} C_DIS
LIN {X -0.036,Y -145.505,Z 1299.196,A 0.000,B 0.000,C 90.000,E1 215.311} C_DIS
LIN {X -0.041,Y -142.909,Z 1299.171,A 0.000,B 0.000,C 90.000,E1 210.718} C_DIS
LIN {X 0.013,Y -141.529,Z 1299.150,A 0.000,B 0.000,C 90.000,E1 207.001} C_DIS
LIN {X 0.056,Y -139.398,Z 1299.114,A 0.000,B 0.000,C 90.000,E1 200.482} C_DIS
LIN {X -0.025,Y -139.111,Z 1299.104,A 0.000,B 0.000,C 90.000,E1 198.652} C_DIS
LIN {X -0.038,Y -138.353,Z 1299.057,A 0.000,B 0.000,C 90.000,E1 190.254} C_DIS
LIN {X -0.048,Y -139.508,Z 1299.005,A 0.000,B 0.000,C 90.000,E1 180.917} C_DIS
LIN {X 0.033,Y -141.147,Z 1298.974,A 0.000,B 0.000,C 90.000,E1 175.298} C_DIS
LIN {X -0.015,Y -142.527,Z 1298.958,A 0.000,B 0.000,C 90.000,E1 172.534} C_DIS
LIN {X -0.069,Y -144.793,Z 1298.933,A 0.000,B 0.000,C 90.000,E1 167.937} C_DIS
LIN {X 0.060,Y -147.411,Z 1298.912,A 0.000,B 0.000,C 90.000,E1 164.212} C_DIS
LIN {X -0.051,Y -149.987,Z 1298.892,A 0.000,B 0.000,C 90.000,E1 160.604} C_DIS
LIN {X -0.042,Y -153.313,Z 1298.872,A 0.000,B 0.000,C 90.000,E1 156.975} C_DIS
LIN {X 0.010,Y -155.014,Z 1298.862,A 0.000,B 0.000,C 90.000,E1 155.153} C_DIS
LIN {X 0.032,Y -158.659,Z 1298.842,A 0.000,B 0.000,C 90.000,E1 151.563} C_DIS
LIN {X -0.024,Y -161.935,Z 1298.827,A 0.000,B 0.000,C 90.000,E1 148.918} C_DIS
LIN {X 0.000,Y -166.126,Z 1298.808,A 0.000,B 0.000,C 90.000,E1 145.388} C_DIS
LIN {X -0.003,Y -171.137,Z 1298.788,A 0.000,B 0.000,C 90.000,E1 141.904} C_DIS
LIN {X 0.032,Y -176.015,Z 1298.769,A 0.000,B 0.000,C 90.000,E1 138.447} C_DIS
LIN {X 0.028,Y -180.266,Z 1298.755,A 0.000,B 0.000,C 90.000,E1 135.891} C_DIS
LIN {X 0.000,Y -185.679,Z 1298.736,A 0.000,B 0.000,C 90.000,E1 132.528} C_DIS
LIN {X 0.053,Y -190.281,Z 1298.722,A 0.000,B 0.000,C 90.000,E1 130.011} C_DIS
LIN {X -0.057,Y -197.608,Z 1298.699,A 0.000,B 0.000,C 90.000,E1 125.931} C_DIS
LIN {X 0.040,Y -199.527,Z 1298.694,A 0.000,B 0.000,C 90.000,E1 124.945} C_DIS
LIN {X 0.026,Y -308.984,Z 1298.694,A 0.000,B 0.000,C 90.000,E1 124.945} C_DIS
LIN {X 0.046,Y -311.408,Z 1298.694,A 0.000,B 0.000,C 90.000,E1 124.898} C_DIS
LIN {X -0.082,Y -316.912,Z 1298.692,A 0.000,B 0.000,C 90.000,E1 124.612} C_DIS
LIN {X 0.052,Y -319.856,Z 1298.690,A 0.000,B 0.000,C 90.000,E1 124.278} C_DIS
LIN {X 0.029,Y -321.864,Z 1298.689,A 0.000,B 0.000,C 90.000,E1 123.992} C_DIS
LIN {X 0.005,Y -323.433,Z 1298.687,A 0.000,B 0.000,C 90.000,E1 123.706} C_DIS
LIN {X 0.093,Y -324.791,Z 1298.686,A 0.000,B 0.000,C 90.000,E1 123.372} C_DIS
LIN {X -0.098,Y -336.427,Z 1298.668,A 0.000,B 0.000,C 90.000,E1 120.256} C_DIS
LIN {X -0.011,Y -348.301,Z 1298.653,A 0.000,B 0.000,C 90.000,E1 117.462} C_DIS
LIN {X 0.119,Y -361.625,Z 1298.637,A 0.000,B 0.000,C 90.000,E1 114.719} C_DIS
LIN {X -0.118,Y -374.782,Z 1298.624,A 0.000,B 0.000,C 90.000,E1 112.386} C_DIS
LIN {X -0.115,Y -389.272,Z 1298.611,A 0.000,B 0.000,C 90.000,E1 110.066} C_DIS
LIN {X 0.135,Y -405.192,Z 1298.599,A 0.000,B 0.000,C 90.000,E1 107.764} C_DIS
LIN {X 0.159,Y -422.659,Z 1298.587,A 0.000,B 0.000,C 90.000,E1 105.552} C_DIS
LIN {X 0.099,Y -441.764,Z 1298.575,A 0.000,B 0.000,C 90.000,E1 103.411} C_DIS
LIN {X -0.080,Y -461.844,Z 1298.563,A 0.000,B 0.000,C 90.000,E1 101.422} C_DIS
LIN {X -0.048,Y -477.233,Z 1298.556,A 0.000,B 0.000,C 90.000,E1 100.018} C_DIS
LIN {X -0.051,Y -479.286,Z 1298.554,A 0.000,B 0.000,C 90.000,E1 99.792} C_DIS
LIN {X -0.177,Y -481.000,Z 1298.553,A 0.000,B 0.000,C 90.000,E1 99.557} C_DIS
LIN {X 0.170,Y -482.285,Z 1298.552,A 0.000,B 0.000,C 90.000,E1 99.265} C_DIS
LIN {X -0.142,Y -483.875,Z 1298.549,A 0.000,B 0.000,C 90.000,E1 98.803} C_DIS
LIN {X 0.103,Y -484.398,Z 1298.546,A 0.000,B 0.000,C 90.000,E1 98.276} C_DIS
LIN {X -0.193,Y -483.946,Z 1298.543,A 0.000,B 0.000,C 90.000,E1 97.814} C_DIS
LIN {X -0.007,Y -482.445,Z 1298.541,A 0.000,B 0.000,C 90.000,E1 97.296} C_DIS
LIN {X -0.183,Y -481.224,Z 1298.539,A 0.000,B 0.000,C 90.000,E1 97.068} C_DIS
LIN {X 0.177,Y -479.595,Z 1298.538,A 0.000,B 0.000,C 90.000,E1 96.777} C_DIS
LIN {X 0.140,Y -468.311,Z 1298.529,A 0.000,B 0.000,C 90.000,E1 95.277} C_DIS
LIN {X -0.113,Y -454.457,Z 1298.518,A 0.000,B 0.000,C 90.000,E1 93.269} C_DIS
LIN {X 0.139,Y -437.801,Z 1298.504,A 0.000,B 0.000,C 90.000,E1 90.630} C_DIS
LIN {X 0.146,Y -420.029,Z 1298.486,A 0.000,B 0.000,C 90.000,E1 87.421} C_DIS
LIN {X 0.105,Y -408.481,Z 1298.474,A 0.000,B 0.000,C 90.000,E1 85.241} C_DIS
LIN {X -0.172,Y -398.204,Z 1298.463,A 0.000,B 0.000,C 90.000,E1 83.337} C_DIS
LIN {X 0.131,Y -387.819,Z 1298.452,A 0.000,B 0.000,C 90.000,E1 81.319} C_DIS
LIN {X -0.085,Y -378.534,Z 1298.442,A 0.000,B 0.000,C 90.000,E1 79.634} C_DIS
LIN {X -0.023,Y -370.605,Z 1298.434,A 0.000,B 0.000,C 90.000,E1 78.173} C_DIS
LIN {X -0.026,Y -360.883,Z 1298.424,A 0.000,B 0.000,C 90.000,E1 76.408} C_DIS
LIN {X -0.173,Y -349.305,Z 1298.413,A 0.000,B 0.000,C 90.000,E1 74.338} C_DIS
LIN {X -0.045,Y -337.697,Z 1298.401,A 0.000,B 0.000,C 90.000,E1 72.181} C_DIS
LIN {X -0.098,Y -324.622,Z 1298.387,A 0.000,B 0.000,C 90.000,E1 69.699} C_DIS
LIN {X 0.011,Y -309.239,Z 1298.369,A 0.000,B 0.000,C 90.000,E1 66.485} C_DIS
LIN {X -0.133,Y -297.874,Z 1298.355,A 0.000,B 0.000,C 90.000,E1 63.896} C_DIS
LIN {X -0.122,Y -290.289,Z 1298.344,A 0.000,B 0.000,C 90.000,E1 61.897} C_DIS
LIN {X -0.142,Y -282.424,Z 1298.331,A 0.000,B 0.000,C 90.000,E1 59.537} C_DIS
LIN {X -0.043,Y -272.409,Z 1298.312,A 0.000,B 0.000,C 90.000,E1 56.087} C_DIS
LIN {X 0.123,Y -263.223,Z 1298.292,A 0.000,B 0.000,C 90.000,E1 52.557} C_DIS
LIN {X -0.013,Y -256.240,Z 1298.276,A 0.000,B 0.000,C 90.000,E1 49.747} C_DIS
LIN {X 0.007,Y -249.457,Z 1298.260,A 0.000,B 0.000,C 90.000,E1 46.863} C_DIS
LIN {X -0.024,Y -241.293,Z 1298.240,A 0.000,B 0.000,C 90.000,E1 43.218} C_DIS
LIN {X 0.068,Y -233.786,Z 1298.219,A 0.000,B 0.000,C 90.000,E1 39.483} C_DIS
LIN {X 0.028,Y -227.193,Z 1298.198,A 0.000,B 0.000,C 90.000,E1 35.724} C_DIS
LIN {X -0.054,Y -221.459,Z 1298.177,A 0.000,B 0.000,C 90.000,E1 31.926} C_DIS
LIN {X 0.091,Y -216.665,Z 1298.156,A 0.000,B 0.000,C 90.000,E1 28.025} C_DIS
LIN {X -0.088,Y -211.567,Z 1298.130,A 0.000,B 0.000,C 90.000,E1 23.387} C_DIS
LIN {X 0.086,Y -207.867,Z 1298.108,A 0.000,B 0.000,C 90.000,E1 19.396} C_DIS
LIN {X -0.004,Y -203.956,Z 1298.081,A 0.000,B 0.000,C 90.000,E1 14.647} C_DIS
LIN {X -0.002,Y -200.360,Z 1298.050,A 0.000,B 0.000,C 90.000,E1 9.029} C_DIS
LIN {X -0.087,Y -197.760,Z 1298.010,A 0.000,B 0.000,C 90.000,E1 1.776} C_DIS
LIN {X -0.038,Y -199.163,Z 1297.943,A 0.000,B 0.000,C 90.000,E1 349.803} C_DIS
LIN {X -0.062,Y -202.575,Z 1297.912,A 0.000,B 0.000,C 90.000,E1 344.157} C_DIS
LIN {X -0.017,Y -206.762,Z 1297.885,A 0.000,B 0.000,C 90.000,E1 339.337} C_DIS
LIN {X 0.016,Y -211.165,Z 1297.863,A 0.000,B 0.000,C 90.000,E1 335.357} C_DIS
LIN {X -0.025,Y -216.269,Z 1297.841,A 0.000,B 0.000,C 90.000,E1 331.435} C_DIS
